Yaskawa INFORM job: A_ROOF_SIDE_0617_2_PAINT_6.JBI

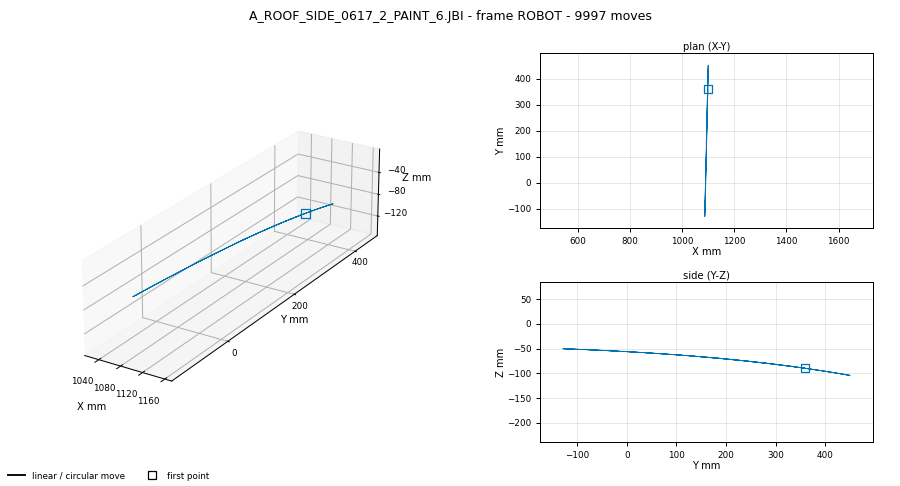
[picture p0: tool path of A_ROOF_SIDE_0617_2_PAINT_6.JBI in frame ROBOT, 9997 of 9997 moves have a stored position in this frame; points joined in program order, loops and branches not executed]
/JOB
//NAME A_ROOF_SIDE_0617_2_PAINT6
//POS
///NPOS 9997,0,0,0,0,0
///TOOL 1
///USER 0
///POSTYPE ROBOT
///RECTAN
///RCONF 1,0,0,0,0,0,0,0,0,0,0,0,0,0,0,0,0,0,0,0,0,0,0,0
C00000=1098.381,359.221,-89.235,178.998,19.661,152.457
C00001=1098.376,358.973,-89.200,178.995,19.657,152.456
C00002=1098.369,358.726,-89.165,178.993,19.653,152.456
C00003=1098.364,358.478,-89.130,178.990,19.649,152.455
C00004=1098.358,358.230,-89.095,178.986,19.645,152.455
C00005=1098.352,357.983,-89.061,178.984,19.641,152.455
C00006=1098.347,357.735,-89.026,178.980,19.637,152.454
C00007=1098.340,357.488,-88.991,178.977,19.632,152.454
C00008=1098.332,357.110,-88.938,178.973,19.626,152.453
C00009=1098.324,356.733,-88.885,178.968,19.620,152.452
C00010=1098.314,356.355,-88.832,178.964,19.614,152.452
C00011=1098.306,355.978,-88.780,178.959,19.608,152.451
C00012=1098.300,355.731,-88.744,178.956,19.604,152.451
C00013=1098.295,355.483,-88.709,178.953,19.600,152.450
C00014=1098.289,355.235,-88.675,178.950,19.596,152.450
C00015=1098.284,354.988,-88.641,178.947,19.592,152.449
C00016=1098.277,354.740,-88.605,178.944,19.588,152.449
C00017=1098.272,354.493,-88.571,178.941,19.585,152.449
C00018=1098.266,354.245,-88.537,178.938,19.580,152.448
C00019=1098.261,353.998,-88.502,178.935,19.576,152.448
C00020=1098.254,353.750,-88.468,178.932,19.572,152.447
C00021=1098.249,353.502,-88.433,178.929,19.568,152.447
C00022=1098.243,353.255,-88.399,178.926,19.565,152.446
C00023=1098.237,353.007,-88.364,178.923,19.561,152.446
C00024=1098.231,352.760,-88.329,178.919,19.557,152.446
C00025=1098.226,352.513,-88.295,178.917,19.553,152.445
C00026=1098.220,352.265,-88.260,178.913,19.549,152.445
C00027=1098.214,352.017,-88.226,178.911,19.545,152.445
C00028=1098.208,351.770,-88.192,178.907,19.541,152.444
C00029=1098.203,351.522,-88.157,178.905,19.538,152.444
C00030=1098.197,351.275,-88.123,178.901,19.534,152.443
C00031=1098.191,351.027,-88.089,178.898,19.530,152.443
C00032=1098.186,350.779,-88.055,178.895,19.526,152.443
C00033=1098.180,350.531,-88.021,178.892,19.522,152.442
C00034=1098.174,350.284,-87.987,178.889,19.519,152.442
C00035=1098.169,350.037,-87.952,178.886,19.515,152.442
C00036=1098.163,349.789,-87.918,178.883,19.512,152.441
C00037=1098.157,349.541,-87.884,178.880,19.507,152.441
C00038=1098.151,349.294,-87.850,178.877,19.504,152.441
C00039=1098.146,349.046,-87.815,178.874,19.500,152.440
C00040=1098.140,348.799,-87.782,178.871,19.497,152.440
C00041=1098.134,348.551,-87.748,178.868,19.493,152.440
C00042=1098.128,348.303,-87.713,178.865,19.489,152.439
C00043=1098.123,348.056,-87.679,178.861,19.485,152.439
C00044=1098.117,347.808,-87.645,178.859,19.482,152.439
C00045=1098.111,347.561,-87.611,178.855,19.478,152.438
C00046=1098.105,347.313,-87.577,178.853,19.475,152.438
C00047=1098.100,347.066,-87.543,178.849,19.470,152.438
C00048=1098.095,346.818,-87.509,178.847,19.467,152.437
C00049=1098.088,346.570,-87.475,178.843,19.463,152.437
C00050=1098.082,346.322,-87.441,178.840,19.460,152.437
C00051=1098.077,346.075,-87.407,178.837,19.456,152.436
C00052=1098.071,345.827,-87.373,178.834,19.453,152.436
C00053=1098.065,345.579,-87.340,178.831,19.449,152.436
C00054=1098.060,345.332,-87.305,178.828,19.445,152.435
C00055=1098.054,345.084,-87.271,178.824,19.442,152.435
C00056=1098.049,344.837,-87.238,178.822,19.438,152.435
C00057=1098.043,344.589,-87.204,178.818,19.434,152.434
C00058=1098.038,344.341,-87.170,178.815,19.431,152.434
C00059=1098.031,344.093,-87.136,178.812,19.427,152.434
C00060=1098.022,343.718,-87.085,178.808,19.422,152.433
C00061=1098.014,343.343,-87.034,178.803,19.417,152.433
C00062=1098.005,342.968,-86.983,178.798,19.412,152.433
C00063=1097.996,342.593,-86.933,178.793,19.406,152.432
C00064=1097.990,342.345,-86.899,178.790,19.403,152.432
C00065=1097.984,342.098,-86.865,178.788,19.400,152.432
C00066=1097.979,341.850,-86.831,178.784,19.396,152.431
C00067=1097.973,341.602,-86.798,178.781,19.393,152.431
C00068=1097.967,341.354,-86.764,178.778,19.389,152.431
C00069=1097.962,341.107,-86.731,178.775,19.386,152.431
C00070=1097.956,340.859,-86.697,178.771,19.382,152.430
C00071=1097.951,340.611,-86.664,178.769,19.379,152.430
C00072=1097.945,340.363,-86.630,178.766,19.376,152.430
C00073=1097.939,340.116,-86.597,178.762,19.372,152.430
C00074=1097.934,339.868,-86.563,178.759,19.369,152.429
C00075=1097.928,339.620,-86.530,178.756,19.365,152.429
C00076=1097.922,339.373,-86.497,178.753,19.362,152.429
C00077=1097.917,339.126,-86.464,178.750,19.359,152.429
C00078=1097.911,338.878,-86.430,178.747,19.355,152.428
C00079=1097.906,338.630,-86.397,178.744,19.352,152.428
C00080=1097.900,338.382,-86.364,178.740,19.349,152.428
C00081=1097.894,338.134,-86.330,178.737,19.345,152.428
C00082=1097.888,337.887,-86.297,178.735,19.342,152.427
C00083=1097.882,337.639,-86.263,178.731,19.339,152.427
C00084=1097.877,337.391,-86.230,178.728,19.335,152.427
C00085=1097.871,337.143,-86.197,178.725,19.332,152.427
C00086=1097.865,336.896,-86.164,178.722,19.329,152.427
C00087=1097.859,336.648,-86.131,178.719,19.326,152.426
C00088=1097.854,336.400,-86.097,178.715,19.322,152.426
C00089=1097.847,336.152,-86.065,178.712,19.319,152.426
C00090=1097.842,335.904,-86.031,178.709,19.316,152.426
C00091=1097.836,335.656,-85.998,178.706,19.312,152.426
C00092=1097.831,335.409,-85.965,178.703,19.309,152.425
C00093=1097.825,335.162,-85.932,178.700,19.307,152.425
C00094=1097.820,334.914,-85.899,178.696,19.303,152.425
C00095=1097.814,334.666,-85.866,178.694,19.300,152.425
C00096=1097.808,334.418,-85.833,178.691,19.297,152.424
C00097=1097.802,334.170,-85.799,178.687,19.293,152.424
C00098=1097.797,333.922,-85.767,178.684,19.290,152.424
C00099=1097.791,333.674,-85.734,178.681,19.287,152.424
C00100=1097.786,333.427,-85.701,178.678,19.283,152.424
C00101=1097.779,333.179,-85.668,178.675,19.281,152.424
C00102=1097.774,332.932,-85.635,178.672,19.278,152.423
C00103=1097.769,332.683,-85.602,178.668,19.274,152.423
C00104=1097.762,332.435,-85.570,178.665,19.271,152.423
C00105=1097.757,332.187,-85.536,178.662,19.268,152.423
C00106=1097.751,331.941,-85.504,178.659,19.265,152.423
C00107=1097.745,331.693,-85.471,178.656,19.262,152.423
C00108=1097.739,331.444,-85.439,178.653,19.259,152.422
C00109=1097.734,331.197,-85.405,178.650,19.256,152.422
C00110=1097.728,330.949,-85.373,178.646,19.253,152.422
C00111=1097.722,330.701,-85.340,178.643,19.250,152.422
C00112=1097.713,330.320,-85.290,178.638,19.245,152.422
C00113=1097.704,329.938,-85.240,178.634,19.240,152.421
C00114=1097.695,329.558,-85.189,178.628,19.236,152.421
C00115=1097.686,329.176,-85.139,178.624,19.231,152.421
C00116=1097.680,328.929,-85.107,178.620,19.228,152.421
C00117=1097.675,328.680,-85.074,178.617,19.225,152.421
C00118=1097.669,328.432,-85.041,178.614,19.222,152.421
C00119=1097.663,328.185,-85.010,178.611,19.220,152.421
C00120=1097.658,327.937,-84.976,178.607,19.216,152.420
C00121=1097.652,327.689,-84.944,178.605,19.213,152.420
C00122=1097.645,327.441,-84.912,178.602,19.211,152.420
C00123=1097.640,327.194,-84.880,178.598,19.208,152.420
C00124=1097.634,326.946,-84.847,178.595,19.204,152.420
C00125=1097.628,326.698,-84.814,178.592,19.201,152.420
C00126=1097.622,326.450,-84.782,178.589,19.199,152.420
C00127=1097.618,326.202,-84.749,178.586,19.196,152.420
C00128=1097.612,325.954,-84.717,178.582,19.193,152.420
C00129=1097.605,325.706,-84.685,178.579,19.190,152.419
C00130=1097.600,325.459,-84.653,178.576,19.187,152.419
C00131=1097.595,325.210,-84.620,178.573,19.184,152.419
C00132=1097.588,324.963,-84.588,178.569,19.181,152.419
C00133=1097.583,324.715,-84.556,178.566,19.178,152.419
C00134=1097.577,324.467,-84.524,178.563,19.175,152.419
C00135=1097.571,324.219,-84.491,178.560,19.173,152.419
C00136=1097.566,323.972,-84.459,178.557,19.170,152.419
C00137=1097.560,323.723,-84.427,178.553,19.167,152.418
C00138=1097.554,323.475,-84.395,178.550,19.164,152.418
C00139=1097.548,323.228,-84.363,178.547,19.161,152.418
C00140=1097.543,322.980,-84.330,178.544,19.158,152.418
C00141=1097.538,322.732,-84.298,178.542,19.155,152.418
C00142=1097.532,322.484,-84.266,178.538,19.152,152.418
C00143=1097.526,322.236,-84.234,178.535,19.149,152.418
C00144=1097.520,321.989,-84.202,178.532,19.147,152.418
C00145=1097.514,321.741,-84.170,178.529,19.144,152.418
C00146=1097.509,321.493,-84.138,178.526,19.141,152.418
C00147=1097.503,321.245,-84.106,178.522,19.138,152.417
C00148=1097.497,320.996,-84.074,178.519,19.135,152.417
C00149=1097.492,320.749,-84.042,178.516,19.133,152.417
C00150=1097.486,320.501,-84.010,178.513,19.130,152.417
C00151=1097.481,320.253,-83.978,178.510,19.127,152.417
C00152=1097.475,320.005,-83.946,178.507,19.125,152.417
C00153=1097.469,319.757,-83.914,178.503,19.121,152.417
C00154=1097.464,319.509,-83.882,178.500,19.119,152.417
C00155=1097.459,319.261,-83.850,178.497,19.116,152.417
C00156=1097.453,319.013,-83.818,178.494,19.113,152.417
C00157=1097.447,318.766,-83.787,178.491,19.111,152.417
C00158=1097.441,318.517,-83.754,178.488,19.108,152.417
C00159=1097.436,318.270,-83.723,178.484,19.105,152.416
C00160=1097.430,318.022,-83.691,178.481,19.102,152.416
C00161=1097.425,317.774,-83.659,178.478,19.099,152.416
C00162=1097.419,317.527,-83.627,178.475,19.097,152.416
C00163=1097.413,317.279,-83.595,178.472,19.094,152.416
C00164=1097.405,316.890,-83.546,178.466,19.089,152.416
C00165=1097.397,316.502,-83.496,178.462,19.085,152.416
C00166=1097.387,316.114,-83.447,178.456,19.081,152.416
C00167=1097.379,315.725,-83.397,178.452,19.077,152.416
C00168=1097.373,315.478,-83.365,178.449,19.074,152.416
C00169=1097.368,315.229,-83.334,178.445,19.071,152.416
C00170=1097.362,314.981,-83.302,178.442,19.068,152.416
C00171=1097.356,314.734,-83.271,178.439,19.066,152.416
C00172=1097.350,314.486,-83.239,178.435,19.063,152.416
C00173=1097.344,314.237,-83.208,178.432,19.061,152.416
C00174=1097.338,313.990,-83.177,178.429,19.058,152.416
C00175=1097.332,313.742,-83.145,178.426,19.056,152.415
C00176=1097.327,313.494,-83.114,178.423,19.053,152.416
C00177=1097.321,313.246,-83.082,178.420,19.051,152.415
C00178=1097.315,312.998,-83.051,178.416,19.047,152.415
C00179=1097.310,312.750,-83.020,178.412,19.045,152.415
C00180=1097.303,312.502,-82.988,178.409,19.043,152.415
C00181=1097.298,312.255,-82.957,178.406,19.040,152.415
C00182=1097.292,312.006,-82.925,178.403,19.038,152.415
C00183=1097.286,311.759,-82.894,178.400,19.035,152.415
C00184=1097.280,311.510,-82.863,178.397,19.033,152.415
C00185=1097.275,311.262,-82.831,178.394,19.030,152.415
C00186=1097.269,311.014,-82.801,178.391,19.028,152.415
C00187=1097.263,310.766,-82.769,178.387,19.025,152.415
C00188=1097.257,310.518,-82.739,178.384,19.023,152.415
C00189=1097.252,310.271,-82.707,178.380,19.020,152.415
C00190=1097.246,310.022,-82.676,178.377,19.017,152.415
C00191=1097.240,309.775,-82.645,178.374,19.015,152.415
C00192=1097.235,309.527,-82.614,178.371,19.013,152.415
C00193=1097.228,309.279,-82.582,178.367,19.010,152.415
C00194=1097.223,309.031,-82.551,178.364,19.008,152.415
C00195=1097.217,308.783,-82.520,178.361,19.005,152.415
C00196=1097.212,308.535,-82.489,178.358,19.003,152.415
C00197=1097.207,308.287,-82.458,178.355,19.000,152.415
C00198=1097.200,308.039,-82.427,178.352,18.998,152.415
C00199=1097.195,307.791,-82.396,178.348,18.996,152.416
C00200=1097.189,307.543,-82.365,178.345,18.993,152.415
C00201=1097.183,307.295,-82.334,178.342,18.991,152.415
C00202=1097.178,307.047,-82.303,178.339,18.988,152.415
C00203=1097.173,306.799,-82.272,178.335,18.985,152.416
C00204=1097.166,306.551,-82.242,178.332,18.983,152.416
C00205=1097.161,306.303,-82.210,178.329,18.980,152.415
C00206=1097.155,306.055,-82.180,178.325,18.978,152.416
C00207=1097.150,305.807,-82.149,178.322,18.975,152.415
C00208=1097.143,305.559,-82.118,178.319,18.973,152.416
C00209=1097.138,305.311,-82.086,178.316,18.971,152.416
C00210=1097.132,305.063,-82.056,178.313,18.968,152.416
C00211=1097.127,304.815,-82.025,178.309,18.966,152.416
C00212=1097.121,304.567,-81.995,178.306,18.963,152.416
C00213=1097.116,304.320,-81.964,178.303,18.961,152.416
C00214=1097.110,304.071,-81.933,178.300,18.958,152.416
C00215=1097.104,303.824,-81.902,178.297,18.956,152.416
C00216=1097.096,303.437,-81.855,178.291,18.952,152.416
C00217=1097.087,303.052,-81.807,178.286,18.948,152.416
C00218=1097.077,302.666,-81.759,178.281,18.945,152.416
C00219=1097.069,302.281,-81.711,178.277,18.941,152.416
C00220=1097.064,302.032,-81.680,178.273,18.939,152.416
C00221=1097.058,301.785,-81.650,178.270,18.936,152.416
C00222=1097.052,301.537,-81.619,178.267,18.934,152.416
C00223=1097.047,301.289,-81.588,178.264,18.932,152.416
C00224=1097.041,301.041,-81.558,178.260,18.928,152.416
C00225=1097.036,300.793,-81.528,178.257,18.926,152.416
C00226=1097.031,300.545,-81.497,178.253,18.924,152.416
C00227=1097.025,300.296,-81.467,178.250,18.922,152.416
C00228=1097.019,300.049,-81.437,178.247,18.919,152.416
C00229=1097.014,299.801,-81.406,178.244,18.917,152.416
C00230=1097.008,299.553,-81.376,178.240,18.914,152.416
C00231=1097.002,299.305,-81.345,178.237,18.912,152.416
C00232=1096.997,299.057,-81.314,178.234,18.910,152.416
C00233=1096.992,298.809,-81.284,178.231,18.907,152.416
C00234=1096.986,298.560,-81.254,178.228,18.905,152.416
C00235=1096.981,298.312,-81.223,178.224,18.903,152.416
C00236=1096.975,298.065,-81.193,178.221,18.900,152.417
C00237=1096.969,297.816,-81.162,178.218,18.898,152.417
C00238=1096.963,297.568,-81.133,178.214,18.896,152.417
C00239=1096.957,297.320,-81.102,178.211,18.894,152.417
C00240=1096.952,297.072,-81.072,178.208,18.891,152.417
C00241=1096.947,296.824,-81.041,178.205,18.889,152.417
C00242=1096.941,296.575,-81.011,178.202,18.887,152.417
C00243=1096.935,296.328,-80.981,178.199,18.885,152.417
C00244=1096.929,296.080,-80.951,178.196,18.883,152.417
C00245=1096.924,295.831,-80.921,178.193,18.880,152.417
C00246=1096.918,295.583,-80.891,178.189,18.878,152.417
C00247=1096.912,295.336,-80.860,178.186,18.876,152.417
C00248=1096.907,295.087,-80.831,178.183,18.874,152.417
C00249=1096.901,294.839,-80.800,178.179,18.871,152.417
C00250=1096.895,294.591,-80.771,178.176,18.869,152.418
C00251=1096.890,294.343,-80.740,178.173,18.867,152.418
C00252=1096.884,294.095,-80.711,178.169,18.865,152.418
C00253=1096.878,293.847,-80.680,178.166,18.863,152.418
C00254=1096.872,293.599,-80.650,178.163,18.860,152.418
C00255=1096.867,293.351,-80.620,178.160,18.858,152.418
C00256=1096.861,293.103,-80.590,178.156,18.856,152.418
C00257=1096.856,292.854,-80.560,178.153,18.854,152.418
C00258=1096.850,292.606,-80.531,178.150,18.851,152.418
C00259=1096.844,292.358,-80.500,178.146,18.849,152.418
C00260=1096.839,292.110,-80.471,178.143,18.847,152.418
C00261=1096.833,291.862,-80.440,178.140,18.845,152.418
C00262=1096.828,291.614,-80.411,178.137,18.842,152.419
C00263=1096.822,291.366,-80.381,178.134,18.841,152.419
C00264=1096.816,291.118,-80.352,178.131,18.839,152.419
C00265=1096.810,290.870,-80.322,178.127,18.837,152.419
C00266=1096.805,290.622,-80.292,178.124,18.834,152.419
C00267=1096.799,290.373,-80.262,178.121,18.832,152.419
C00268=1096.791,290.001,-80.217,178.116,18.829,152.419
C00269=1096.782,289.630,-80.173,178.111,18.826,152.419
C00270=1096.774,289.258,-80.128,178.106,18.822,152.420
C00271=1096.765,288.887,-80.084,178.101,18.819,152.420
C00272=1096.759,288.638,-80.054,178.098,18.817,152.420
C00273=1096.754,288.390,-80.025,178.095,18.815,152.420
C00274=1096.748,288.141,-79.995,178.092,18.813,152.420
C00275=1096.742,287.894,-79.965,178.088,18.811,152.420
C00276=1096.736,287.645,-79.936,178.085,18.809,152.420
C00277=1096.731,287.398,-79.906,178.082,18.807,152.420
C00278=1096.726,287.149,-79.877,178.078,18.805,152.420
C00279=1096.720,286.901,-79.848,178.075,18.802,152.421
C00280=1096.714,286.653,-79.818,178.071,18.801,152.421
C00281=1096.709,286.404,-79.789,178.068,18.798,152.421
C00282=1096.702,286.157,-79.759,178.066,18.797,152.421
C00283=1096.697,285.909,-79.730,178.062,18.794,152.421
C00284=1096.692,285.660,-79.700,178.059,18.793,152.421
C00285=1096.685,285.412,-79.671,178.056,18.790,152.421
C00286=1096.680,285.164,-79.641,178.052,18.788,152.421
C00287=1096.674,284.915,-79.612,178.049,18.786,152.422
C00288=1096.669,284.668,-79.583,178.046,18.784,152.422
C00289=1096.663,284.420,-79.553,178.042,18.782,152.422
C00290=1096.658,284.171,-79.524,178.040,18.780,152.422
C00291=1096.651,283.923,-79.495,178.036,18.778,152.422
C00292=1096.646,283.675,-79.465,178.033,18.776,152.422
C00293=1096.641,283.427,-79.436,178.030,18.774,152.422
C00294=1096.635,283.179,-79.407,178.026,18.772,152.422
C00295=1096.629,282.930,-79.377,178.023,18.770,152.423
C00296=1096.624,282.681,-79.348,178.020,18.767,152.423
C00297=1096.618,282.434,-79.319,178.016,18.766,152.423
C00298=1096.613,282.185,-79.290,178.014,18.764,152.423
C00299=1096.607,281.937,-79.261,178.010,18.762,152.423
C00300=1096.602,281.689,-79.231,178.007,18.760,152.423
C00301=1096.595,281.441,-79.202,178.004,18.758,152.423
C00302=1096.590,281.193,-79.173,178.000,18.755,152.423
C00303=1096.584,280.944,-79.144,177.997,18.754,152.424
C00304=1096.579,280.696,-79.115,177.994,18.751,152.424
C00305=1096.573,280.448,-79.086,177.991,18.750,152.424
C00306=1096.567,280.200,-79.057,177.988,18.748,152.424
C00307=1096.561,279.951,-79.028,177.984,18.746,152.424
C00308=1096.556,279.703,-78.999,177.981,18.744,152.424
C00309=1096.550,279.455,-78.970,177.977,18.741,152.424
C00310=1096.545,279.207,-78.940,177.974,18.740,152.425
C00311=1096.539,278.959,-78.912,177.971,18.738,152.425
C00312=1096.533,278.711,-78.883,177.968,18.736,152.425
C00313=1096.528,278.462,-78.854,177.965,18.734,152.425
C00314=1096.522,278.214,-78.826,177.961,18.732,152.425
C00315=1096.517,277.966,-78.796,177.958,18.730,152.425
C00316=1096.511,277.717,-78.768,177.954,18.728,152.426
C00317=1096.505,277.469,-78.739,177.952,18.726,152.426
C00318=1096.500,277.221,-78.709,177.948,18.724,152.426
C00319=1096.494,276.972,-78.681,177.945,18.722,152.426
C00320=1096.486,276.610,-78.639,177.940,18.719,152.426
C00321=1096.478,276.248,-78.597,177.936,18.717,152.427
C00322=1096.469,275.885,-78.555,177.931,18.714,152.427
C00323=1096.460,275.523,-78.513,177.926,18.711,152.427
C00324=1096.456,275.275,-78.485,177.923,18.709,152.427
C00325=1096.450,275.026,-78.455,177.920,18.707,152.427
C00326=1096.444,274.778,-78.427,177.916,18.705,152.427
C00327=1096.439,274.530,-78.398,177.913,18.703,152.428
C00328=1096.433,274.281,-78.370,177.910,18.702,152.428
C00329=1096.427,274.034,-78.341,177.907,18.700,152.428
C00330=1096.421,273.785,-78.313,177.903,18.698,152.428
C00331=1096.416,273.536,-78.284,177.900,18.696,152.428
C00332=1096.410,273.289,-78.255,177.896,18.694,152.428
C00333=1096.404,273.040,-78.227,177.894,18.692,152.429
C00334=1096.399,272.792,-78.198,177.890,18.690,152.429
C00335=1096.393,272.544,-78.170,177.887,18.688,152.429
C00336=1096.388,272.295,-78.141,177.884,18.686,152.429
C00337=1096.382,272.046,-78.113,177.881,18.685,152.429
C00338=1096.376,271.798,-78.084,177.877,18.683,152.430
C00339=1096.371,271.550,-78.056,177.874,18.681,152.430
C00340=1096.365,271.302,-78.027,177.871,18.679,152.430
C00341=1096.359,271.054,-77.999,177.867,18.677,152.430
C00342=1096.353,270.805,-77.970,177.865,18.676,152.430
C00343=1096.349,270.557,-77.942,177.861,18.674,152.430
C00344=1096.343,270.308,-77.914,177.858,18.671,152.430
C00345=1096.337,270.060,-77.886,177.854,18.670,152.431
C00346=1096.331,269.812,-77.857,177.852,18.668,152.431
C00347=1096.326,269.564,-77.829,177.848,18.666,152.431
C00348=1096.320,269.315,-77.800,177.845,18.664,152.431
C00349=1096.314,269.067,-77.772,177.841,18.663,152.431
C00350=1096.308,268.818,-77.744,177.838,18.660,152.432
C00351=1096.303,268.570,-77.716,177.835,18.659,152.432
C00352=1096.297,268.322,-77.688,177.832,18.657,152.432
C00353=1096.292,268.074,-77.659,177.828,18.655,152.432
C00354=1096.286,267.825,-77.631,177.825,18.653,152.432
C00355=1096.280,267.577,-77.603,177.822,18.652,152.433
C00356=1096.274,267.329,-77.574,177.819,18.650,152.433
C00357=1096.269,267.081,-77.546,177.815,18.648,152.433
C00358=1096.263,266.832,-77.518,177.812,18.646,152.433
C00359=1096.258,266.584,-77.490,177.809,18.644,152.433
C00360=1096.252,266.335,-77.462,177.806,18.643,152.433
C00361=1096.246,266.087,-77.434,177.802,18.641,152.434
C00362=1096.241,265.839,-77.406,177.799,18.639,152.434
C00363=1096.235,265.590,-77.378,177.796,18.637,152.434
C00364=1096.230,265.342,-77.350,177.793,18.636,152.434
C00365=1096.224,265.093,-77.322,177.789,18.634,152.434
C00366=1096.219,264.845,-77.294,177.786,18.631,152.435
C00367=1096.213,264.597,-77.266,177.783,18.630,152.435
C00368=1096.207,264.348,-77.238,177.780,18.628,152.435
C00369=1096.201,264.100,-77.210,177.776,18.627,152.435
C00370=1096.195,263.851,-77.182,177.773,18.625,152.435
C00371=1096.190,263.603,-77.154,177.770,18.623,152.436
C00372=1096.182,263.243,-77.115,177.765,18.621,152.436
C00373=1096.173,262.884,-77.074,177.760,18.618,152.436
C00374=1096.165,262.525,-77.034,177.756,18.616,152.437
C00375=1096.157,262.164,-76.994,177.751,18.613,152.437
C00376=1096.151,261.916,-76.966,177.748,18.612,152.437
C00377=1096.145,261.668,-76.938,177.745,18.610,152.437
C00378=1096.139,261.420,-76.910,177.741,18.608,152.438
C00379=1096.134,261.171,-76.883,177.738,18.606,152.438
C00380=1096.128,260.923,-76.855,177.735,18.605,152.438
C00381=1096.122,260.674,-76.827,177.731,18.603,152.438
C00382=1096.116,260.426,-76.799,177.728,18.602,152.439
C00383=1096.111,260.178,-76.772,177.725,18.600,152.439
C00384=1096.105,259.929,-76.744,177.722,18.598,152.439
C00385=1096.100,259.680,-76.717,177.718,18.596,152.439
C00386=1096.094,259.432,-76.689,177.716,18.595,152.439
C00387=1096.088,259.184,-76.661,177.712,18.593,152.440
C00388=1096.083,258.935,-76.634,177.709,18.591,152.440
C00389=1096.076,258.687,-76.606,177.705,18.590,152.440
C00390=1096.071,258.438,-76.579,177.702,18.588,152.440
C00391=1096.065,258.190,-76.551,177.699,18.586,152.440
C00392=1096.060,257.942,-76.524,177.695,18.584,152.441
C00393=1096.054,257.693,-76.496,177.693,18.583,152.441
C00394=1096.048,257.445,-76.469,177.689,18.581,152.441
C00395=1096.043,257.196,-76.441,177.686,18.580,152.441
C00396=1096.037,256.948,-76.415,177.683,18.578,152.442
C00397=1096.031,256.699,-76.386,177.679,18.576,152.442
C00398=1096.026,256.451,-76.359,177.676,18.575,152.442
C00399=1096.020,256.203,-76.332,177.673,18.573,152.442
C00400=1096.015,255.954,-76.305,177.670,18.571,152.442
C00401=1096.008,255.706,-76.277,177.666,18.569,152.443
C00402=1096.003,255.457,-76.250,177.664,18.568,152.443
C00403=1095.997,255.209,-76.223,177.660,18.566,152.443
C00404=1095.992,254.961,-76.195,177.657,18.565,152.443
C00405=1095.986,254.712,-76.168,177.654,18.563,152.444
C00406=1095.980,254.464,-76.140,177.650,18.562,152.444
C00407=1095.974,254.215,-76.113,177.647,18.560,152.444
C00408=1095.969,253.966,-76.086,177.644,18.558,152.444
C00409=1095.963,253.719,-76.059,177.641,18.556,152.444
C00410=1095.958,253.469,-76.031,177.637,18.554,152.445
C00411=1095.952,253.221,-76.004,177.635,18.553,152.445
C00412=1095.947,252.972,-75.977,177.631,18.551,152.445
C00413=1095.941,252.725,-75.950,177.628,18.550,152.445
C00414=1095.936,252.476,-75.923,177.625,18.548,152.446
C00415=1095.930,252.228,-75.896,177.621,18.547,152.446
C00416=1095.924,251.978,-75.868,177.618,18.544,152.446
C00417=1095.919,251.730,-75.842,177.615,18.543,152.446
C00418=1095.913,251.482,-75.814,177.612,18.541,152.446
C00419=1095.908,251.233,-75.787,177.608,18.540,152.447
C00420=1095.902,250.985,-75.760,177.606,18.538,152.447
C00421=1095.897,250.736,-75.733,177.602,18.536,152.447
C00422=1095.892,250.488,-75.706,177.598,18.535,152.447
C00423=1095.886,250.239,-75.679,177.596,18.533,152.448
C00424=1095.877,249.877,-75.639,177.591,18.531,152.448
C00425=1095.869,249.514,-75.600,177.586,18.528,152.448
C00426=1095.862,249.152,-75.561,177.582,18.526,152.448
C00427=1095.853,248.789,-75.521,177.576,18.523,152.449
C00428=1095.847,248.540,-75.494,177.574,18.522,152.449
C00429=1095.842,248.292,-75.468,177.570,18.520,152.449
C00430=1095.837,248.043,-75.441,177.567,18.518,152.449
C00431=1095.831,247.795,-75.414,177.564,18.517,152.450
C00432=1095.826,247.546,-75.387,177.561,18.515,152.450
C00433=1095.820,247.298,-75.360,177.558,18.514,152.450
C00434=1095.814,247.050,-75.333,177.554,18.512,152.450
C00435=1095.809,246.801,-75.307,177.551,18.510,152.451
C00436=1095.804,246.553,-75.279,177.548,18.509,152.451
C00437=1095.798,246.304,-75.253,177.545,18.507,152.451
C00438=1095.792,246.055,-75.227,177.541,18.505,152.451
C00439=1095.786,245.807,-75.200,177.538,18.504,152.452
C00440=1095.781,245.559,-75.174,177.535,18.502,152.452
C00441=1095.776,245.310,-75.146,177.532,18.501,152.452
C00442=1095.770,245.062,-75.120,177.529,18.499,152.452
C00443=1095.764,244.813,-75.093,177.525,18.498,152.453
C00444=1095.758,244.565,-75.066,177.522,18.496,152.453
C00445=1095.753,244.316,-75.040,177.519,18.495,152.453
C00446=1095.748,244.067,-75.013,177.516,18.493,152.453
C00447=1095.742,243.819,-74.987,177.513,18.492,152.454
C00448=1095.736,243.570,-74.960,177.509,18.490,152.454
C00449=1095.731,243.321,-74.934,177.506,18.489,152.454
C00450=1095.725,243.073,-74.907,177.503,18.487,152.454
C00451=1095.719,242.825,-74.881,177.500,18.486,152.454
C00452=1095.714,242.576,-74.854,177.497,18.484,152.455
C00453=1095.708,242.327,-74.828,177.493,18.482,152.455
C00454=1095.702,242.079,-74.801,177.490,18.481,152.455
C00455=1095.697,241.831,-74.775,177.487,18.479,152.455
C00456=1095.691,241.582,-74.749,177.484,18.478,152.456
C00457=1095.685,241.333,-74.722,177.481,18.476,152.456
C00458=1095.679,241.085,-74.696,177.478,18.475,152.456
C00459=1095.674,240.836,-74.670,177.474,18.473,152.456
C00460=1095.668,240.588,-74.643,177.471,18.471,152.457
C00461=1095.663,240.339,-74.617,177.468,18.470,152.457
C00462=1095.657,240.090,-74.590,177.465,18.468,152.457
C00463=1095.651,239.842,-74.564,177.462,18.467,152.457
C00464=1095.646,239.593,-74.538,177.458,18.466,152.458
C00465=1095.640,239.345,-74.511,177.454,18.464,152.458
C00466=1095.635,239.096,-74.485,177.452,18.462,152.458
C00467=1095.629,238.847,-74.459,177.448,18.461,152.459
C00468=1095.623,238.598,-74.433,177.446,18.459,152.459
C00469=1095.618,238.350,-74.406,177.442,18.458,152.459
C00470=1095.613,238.102,-74.380,177.439,18.456,152.459
C00471=1095.607,237.853,-74.354,177.436,18.455,152.460
C00472=1095.601,237.604,-74.328,177.433,18.453,152.460
C00473=1095.595,237.356,-74.302,177.429,18.452,152.460
C00474=1095.589,237.107,-74.276,177.426,18.450,152.460
C00475=1095.584,236.858,-74.250,177.423,18.449,152.460
C00476=1095.576,236.489,-74.211,177.419,18.447,152.461
C00477=1095.567,236.120,-74.173,177.413,18.444,152.461
C00478=1095.559,235.751,-74.133,177.409,18.442,152.462
C00479=1095.551,235.381,-74.095,177.404,18.440,152.462
C00480=1095.545,235.133,-74.069,177.401,18.438,152.462
C00481=1095.540,234.884,-74.043,177.398,18.437,152.463
C00482=1095.534,234.635,-74.017,177.394,18.435,152.463
C00483=1095.529,234.386,-73.991,177.392,18.434,152.463
C00484=1095.523,234.138,-73.965,177.388,18.432,152.463
C00485=1095.517,233.889,-73.939,177.385,18.431,152.464
C00486=1095.512,233.640,-73.913,177.382,18.429,152.464
C00487=1095.506,233.392,-73.887,177.378,18.427,152.464
C00488=1095.500,233.143,-73.861,177.375,18.427,152.464
C00489=1095.495,232.895,-73.836,177.372,18.425,152.465
C00490=1095.489,232.646,-73.810,177.369,18.424,152.465
C00491=1095.484,232.397,-73.784,177.366,18.422,152.465
C00492=1095.478,232.149,-73.758,177.363,18.421,152.465
C00493=1095.472,231.900,-73.732,177.359,18.419,152.466
C00494=1095.467,231.652,-73.706,177.357,18.418,152.466
C00495=1095.461,231.403,-73.681,177.353,18.416,152.466
C00496=1095.456,231.154,-73.655,177.350,18.415,152.466
C00497=1095.450,230.905,-73.629,177.347,18.413,152.467
C00498=1095.445,230.657,-73.603,177.344,18.412,152.467
C00499=1095.439,230.408,-73.578,177.340,18.410,152.467
C00500=1095.433,230.159,-73.552,177.338,18.409,152.468
C00501=1095.427,229.911,-73.526,177.334,18.407,152.468
C00502=1095.422,229.663,-73.501,177.331,18.406,152.468
C00503=1095.416,229.414,-73.475,177.328,18.404,152.468
C00504=1095.410,229.165,-73.449,177.325,18.404,152.469
C00505=1095.404,228.917,-73.424,177.321,18.402,152.469
C00506=1095.399,228.668,-73.398,177.319,18.401,152.469
C00507=1095.394,228.419,-73.372,177.315,18.399,152.469
C00508=1095.388,228.171,-73.347,177.312,18.398,152.470
C00509=1095.382,227.922,-73.321,177.309,18.396,152.470
C00510=1095.377,227.674,-73.296,177.306,18.395,152.470
C00511=1095.371,227.425,-73.270,177.302,18.393,152.471
C00512=1095.365,227.176,-73.246,177.300,18.392,152.471
C00513=1095.360,226.927,-73.220,177.296,18.390,152.471
C00514=1095.354,226.679,-73.195,177.293,18.389,152.471
C00515=1095.349,226.430,-73.169,177.290,18.387,152.472
C00516=1095.343,226.182,-73.144,177.287,18.386,152.472
C00517=1095.337,225.933,-73.119,177.283,18.385,152.472
C00518=1095.331,225.684,-73.093,177.281,18.383,152.472
C00519=1095.326,225.436,-73.068,177.277,18.382,152.473
C00520=1095.321,225.186,-73.042,177.274,18.380,152.473
C00521=1095.314,224.938,-73.017,177.271,18.379,152.473
C00522=1095.310,224.689,-72.991,177.268,18.378,152.474
C00523=1095.303,224.441,-72.966,177.264,18.376,152.474
C00524=1095.298,224.192,-72.940,177.262,18.375,152.474
C00525=1095.293,223.943,-72.916,177.258,18.373,152.474
C00526=1095.286,223.695,-72.891,177.255,18.372,152.475
C00527=1095.282,223.446,-72.865,177.252,18.370,152.475
C00528=1095.273,223.068,-72.826,177.247,18.368,152.475
C00529=1095.265,222.689,-72.789,177.243,18.366,152.476
C00530=1095.256,222.312,-72.750,177.238,18.364,152.476
C00531=1095.247,221.934,-72.712,177.233,18.362,152.477
C00532=1095.242,221.685,-72.686,177.230,18.360,152.477
C00533=1095.236,221.436,-72.662,177.227,18.360,152.477
C00534=1095.230,221.188,-72.637,177.224,18.358,152.477
C00535=1095.225,220.940,-72.612,177.221,18.357,152.478
C00536=1095.219,220.690,-72.586,177.217,18.355,152.478
C00537=1095.213,220.442,-72.561,177.214,18.354,152.478
C00538=1095.208,220.193,-72.537,177.211,18.352,152.479
C00539=1095.202,219.944,-72.512,177.208,18.351,152.479
C00540=1095.197,219.695,-72.487,177.205,18.349,152.479
C00541=1095.191,219.447,-72.461,177.202,18.348,152.479
C00542=1095.186,219.198,-72.437,177.198,18.347,152.480
C00543=1095.179,218.949,-72.412,177.195,18.345,152.480
C00544=1095.174,218.701,-72.388,177.193,18.344,152.480
C00545=1095.169,218.452,-72.362,177.189,18.342,152.480
C00546=1095.163,218.203,-72.337,177.186,18.342,152.481
C00547=1095.157,217.955,-72.312,177.183,18.340,152.481
C00548=1095.151,217.705,-72.287,177.180,18.339,152.481
C00549=1095.146,217.457,-72.262,177.176,18.337,152.482
C00550=1095.140,217.208,-72.238,177.174,18.336,152.482
C00551=1095.135,216.960,-72.212,177.171,18.335,152.482
C00552=1095.130,216.711,-72.188,177.167,18.333,152.483
C00553=1095.124,216.462,-72.163,177.164,18.332,152.483
C00554=1095.118,216.214,-72.138,177.161,18.330,152.483
C00555=1095.112,215.965,-72.114,177.158,18.329,152.483
C00556=1095.107,215.717,-72.089,177.154,18.328,152.484
C00557=1095.101,215.467,-72.064,177.152,18.326,152.484
C00558=1095.095,215.219,-72.040,177.149,18.325,152.484
C00559=1095.090,214.970,-72.014,177.145,18.323,152.484
C00560=1095.085,214.721,-71.990,177.143,18.322,152.485
C00561=1095.079,214.473,-71.965,177.139,18.321,152.485
C00562=1095.073,214.223,-71.941,177.136,18.320,152.485
C00563=1095.068,213.975,-71.916,177.133,18.319,152.486
C00564=1095.062,213.726,-71.891,177.130,18.317,152.486
C00565=1095.057,213.478,-71.867,177.127,18.316,152.486
C00566=1095.051,213.229,-71.843,177.124,18.314,152.486
C00567=1095.045,212.980,-71.817,177.121,18.313,152.487
C00568=1095.040,212.732,-71.793,177.118,18.312,152.487
C00569=1095.034,212.482,-71.768,177.114,18.310,152.487
C00570=1095.029,212.234,-71.744,177.112,18.309,152.487
C00571=1095.023,211.985,-71.720,177.108,18.307,152.488
C00572=1095.017,211.737,-71.695,177.105,18.306,152.488
C00573=1095.012,211.488,-71.670,177.102,18.305,152.488
C00574=1095.006,211.239,-71.646,177.099,18.303,152.489
C00575=1095.001,210.990,-71.622,177.096,18.302,152.489
C00576=1094.995,210.742,-71.597,177.092,18.301,152.489
C00577=1094.989,210.492,-71.573,177.090,18.300,152.490
C00578=1094.984,210.244,-71.548,177.087,18.298,152.490
C00579=1094.978,209.995,-71.525,177.083,18.297,152.490
C00580=1094.970,209.621,-71.488,177.079,18.295,152.490
C00581=1094.961,209.247,-71.451,177.074,18.293,152.491
C00582=1094.952,208.872,-71.415,177.070,18.291,152.491
C00583=1094.944,208.498,-71.378,177.065,18.289,152.492
C00584=1094.921,207.483,-71.280,177.011,18.266,152.497
C00585=1094.916,207.234,-71.256,177.008,18.266,152.497
C00586=1094.910,206.986,-71.232,177.005,18.265,152.498
C00587=1094.904,206.737,-71.207,177.002,18.265,152.498
C00588=1094.899,206.488,-71.184,176.998,18.264,152.499
C00589=1094.893,206.239,-71.160,176.995,18.264,152.499
C00590=1094.888,205.991,-71.136,176.991,18.263,152.500
C00591=1094.882,205.741,-71.111,176.988,18.262,152.500
C00592=1094.876,205.492,-71.088,176.985,18.262,152.501
C00593=1094.871,205.244,-71.064,176.982,18.262,152.501
C00594=1094.865,204.996,-71.040,176.979,18.261,152.502
C00595=1094.860,204.746,-71.017,176.975,18.261,152.502
C00596=1094.855,204.498,-70.993,176.972,18.261,152.503
C00597=1094.848,204.249,-70.969,176.969,18.260,152.503
C00598=1094.843,204.000,-70.945,176.966,18.260,152.504
C00599=1094.837,203.751,-70.921,176.963,18.259,152.504
C00600=1094.832,203.503,-70.897,176.960,18.259,152.505
C00601=1094.827,203.254,-70.874,176.956,18.258,152.505
C00602=1094.821,203.005,-70.850,176.953,18.258,152.506
C00603=1094.816,202.756,-70.826,176.949,18.257,152.506
C00604=1094.809,202.507,-70.802,176.946,18.256,152.507
C00605=1094.804,202.258,-70.779,176.943,18.256,152.507
C00606=1094.798,202.010,-70.755,176.940,18.256,152.508
C00607=1094.792,201.761,-70.732,176.937,18.255,152.508
C00608=1094.787,201.512,-70.708,176.933,18.255,152.509
C00609=1094.780,201.263,-70.684,176.930,18.255,152.509
C00610=1094.775,201.014,-70.660,176.927,18.254,152.510
C00611=1094.769,200.766,-70.637,176.924,18.254,152.510
C00612=1094.764,200.517,-70.614,176.921,18.253,152.511
C00613=1094.758,200.268,-70.590,176.917,18.253,152.511
C00614=1094.752,200.019,-70.567,176.914,18.253,152.512
C00615=1094.747,199.770,-70.544,176.911,18.252,152.512
C00616=1094.741,199.521,-70.519,176.908,18.252,152.513
C00617=1094.735,199.272,-70.496,176.905,18.251,152.514
C00618=1094.729,199.024,-70.472,176.902,18.251,152.514
C00619=1094.724,198.775,-70.449,176.898,18.250,152.514
C00620=1094.718,198.526,-70.426,176.895,18.250,152.515
C00621=1094.712,198.278,-70.402,176.892,18.249,152.515
C00622=1094.707,198.028,-70.379,176.889,18.249,152.516
C00623=1094.701,197.780,-70.355,176.886,18.249,152.517
C00624=1094.696,197.531,-70.332,176.882,18.248,152.517
C00625=1094.691,197.282,-70.309,176.879,18.247,152.517
C00626=1094.685,197.034,-70.285,176.875,18.247,152.518
C00627=1094.678,196.784,-70.262,176.872,18.246,152.518
C00628=1094.673,196.535,-70.238,176.869,18.246,152.519
C00629=1094.667,196.286,-70.215,176.866,18.245,152.519
C00630=1094.661,196.038,-70.191,176.863,18.245,152.520
C00631=1094.656,195.788,-70.168,176.860,18.245,152.520
C00632=1094.651,195.540,-70.145,176.857,18.244,152.521
C00633=1094.645,195.291,-70.122,176.853,18.244,152.521
C00634=1094.639,195.042,-70.098,176.851,18.243,152.522
C00635=1094.634,194.793,-70.075,176.847,18.243,152.522
C00636=1094.628,194.544,-70.052,176.844,18.243,152.523
C00637=1094.622,194.295,-70.029,176.841,18.242,152.523
C00638=1094.617,194.047,-70.006,176.838,18.242,152.524
C00639=1094.611,193.798,-69.982,176.835,18.241,152.524
C00640=1094.606,193.549,-69.959,176.832,18.241,152.525
C00641=1094.600,193.300,-69.936,176.829,18.240,152.525
C00642=1094.594,193.051,-69.913,176.825,18.240,152.526
C00643=1094.589,192.802,-69.889,176.822,18.239,152.526
C00644=1094.584,192.553,-69.866,176.819,18.239,152.527
C00645=1094.577,192.278,-69.841,176.816,18.238,152.527
C00646=1094.572,192.003,-69.816,176.812,18.237,152.528
C00647=1094.565,191.729,-69.790,176.809,18.237,152.528
C00648=1094.559,191.453,-69.765,176.806,18.237,152.529
C00649=1094.553,191.204,-69.742,176.803,18.236,152.529
C00650=1094.548,190.955,-69.719,176.799,18.236,152.530
C00651=1094.543,190.706,-69.695,176.796,18.235,152.530
C00652=1094.537,190.457,-69.672,176.793,18.235,152.531
C00653=1094.531,190.208,-69.649,176.790,18.234,152.531
C00654=1094.526,189.959,-69.626,176.787,18.234,152.532
C00655=1094.520,189.710,-69.603,176.784,18.233,152.532
C00656=1094.515,189.462,-69.581,176.781,18.233,152.533
C00657=1094.510,189.213,-69.557,176.778,18.232,152.533
C00658=1094.504,188.964,-69.534,176.774,18.232,152.534
C00659=1094.498,188.715,-69.511,176.771,18.231,152.534
C00660=1094.493,188.466,-69.488,176.768,18.230,152.534
C00661=1094.487,188.217,-69.465,176.765,18.230,152.535
C00662=1094.481,187.968,-69.443,176.762,18.229,152.535
C00663=1094.476,187.720,-69.420,176.759,18.229,152.536
C00664=1094.471,187.471,-69.396,176.756,18.228,152.536
C00665=1094.465,187.222,-69.373,176.753,18.228,152.537
C00666=1094.460,186.973,-69.351,176.750,18.227,152.537
C00667=1094.454,186.724,-69.328,176.747,18.227,152.538
C00668=1094.449,186.476,-69.306,176.744,18.226,152.538
C00669=1094.443,186.227,-69.283,176.740,18.226,152.539
C00670=1094.437,185.978,-69.260,176.737,18.225,152.539
C00671=1094.432,185.729,-69.237,176.734,18.224,152.539
C00672=1094.426,185.479,-69.215,176.731,18.224,152.540
C00673=1094.421,185.231,-69.192,176.728,18.223,152.540
C00674=1094.415,184.982,-69.169,176.725,18.223,152.541
C00675=1094.410,184.733,-69.146,176.722,18.222,152.541
C00676=1094.404,184.484,-69.124,176.719,18.222,152.542
C00677=1094.399,184.235,-69.101,176.716,18.221,152.542
C00678=1094.392,183.986,-69.079,176.713,18.221,152.543
C00679=1094.386,183.737,-69.056,176.710,18.220,152.543
C00680=1094.381,183.488,-69.033,176.706,18.220,152.544
C00681=1094.375,183.239,-69.010,176.703,18.219,152.544
C00682=1094.370,182.991,-68.988,176.700,18.219,152.545
C00683=1094.364,182.742,-68.966,176.697,18.218,152.545
C00684=1094.358,182.493,-68.943,176.694,18.218,152.545
C00685=1094.352,182.244,-68.920,176.692,18.218,152.546
C00686=1094.347,181.995,-68.897,176.689,18.217,152.546
C00687=1094.341,181.746,-68.876,176.685,18.217,152.547
C00688=1094.335,181.498,-68.853,176.682,18.216,152.547
C00689=1094.330,181.248,-68.831,176.679,18.216,152.548
C00690=1094.324,180.999,-68.808,176.676,18.215,152.548
C00691=1094.318,180.751,-68.786,176.673,18.215,152.549
C00692=1094.312,180.501,-68.763,176.670,18.214,152.549
C00693=1094.307,180.252,-68.741,176.667,18.213,152.550
C00694=1094.301,180.004,-68.719,176.664,18.213,152.550
C00695=1094.295,179.755,-68.696,176.661,18.213,152.551
C00696=1094.290,179.505,-68.674,176.657,18.212,152.551
C00697=1094.283,179.257,-68.652,176.654,18.212,152.552
C00698=1094.278,179.008,-68.629,176.651,18.211,152.552
C00699=1094.273,178.759,-68.607,176.648,18.211,152.553
C00700=1094.267,178.510,-68.584,176.645,18.210,152.553
C00701=1094.261,178.261,-68.562,176.642,18.209,152.553
C00702=1094.256,178.012,-68.540,176.640,18.209,152.554
C00703=1094.250,177.763,-68.518,176.637,18.209,152.554
C00704=1094.244,177.514,-68.496,176.634,18.208,152.555
C00705=1094.239,177.265,-68.473,176.631,18.208,152.555
C00706=1094.233,177.017,-68.452,176.628,18.207,152.556
C00707=1094.227,176.768,-68.429,176.625,18.206,152.556
C00708=1094.222,176.518,-68.407,176.621,18.206,152.557
C00709=1094.215,176.243,-68.382,176.618,18.205,152.557
C00710=1094.210,175.967,-68.358,176.615,18.205,152.558
C00711=1094.203,175.692,-68.333,176.611,18.204,152.558
C00712=1094.197,175.416,-68.309,176.608,18.204,152.559
C00713=1094.191,175.167,-68.286,176.605,18.203,152.559
C00714=1094.185,174.918,-68.264,176.602,18.202,152.559
C00715=1094.181,174.669,-68.242,176.599,18.202,152.560
C00716=1094.174,174.421,-68.220,176.596,18.201,152.560
C00717=1094.169,174.172,-68.198,176.593,18.201,152.561
C00718=1094.163,173.922,-68.176,176.591,18.200,152.561
C00719=1094.157,173.674,-68.153,176.588,18.200,152.562
C00720=1094.153,173.425,-68.132,176.585,18.199,152.562
C00721=1094.146,173.176,-68.110,176.581,18.199,152.562
C00722=1094.141,172.926,-68.088,176.578,18.198,152.563
C00723=1094.135,172.678,-68.066,176.575,18.197,152.563
C00724=1094.130,172.429,-68.043,176.572,18.197,152.564
C00725=1094.124,172.179,-68.022,176.569,18.196,152.564
C00726=1094.119,171.931,-68.000,176.566,18.195,152.565
C00727=1094.112,171.682,-67.978,176.563,18.195,152.565
C00728=1094.107,171.433,-67.956,176.561,18.195,152.565
C00729=1094.102,171.184,-67.934,176.558,18.194,152.566
C00730=1094.096,170.935,-67.912,176.555,18.193,152.566
C00731=1094.091,170.686,-67.890,176.552,18.193,152.567
C00732=1094.085,170.436,-67.868,176.549,18.192,152.567
C00733=1094.080,170.188,-67.847,176.546,18.191,152.567
C00734=1094.074,169.939,-67.824,176.543,18.191,152.568
C00735=1094.069,169.690,-67.802,176.540,18.190,152.568
C00736=1094.063,169.441,-67.781,176.537,18.190,152.569
C00737=1094.058,169.192,-67.759,176.534,18.189,152.569
C00738=1094.052,168.943,-67.737,176.532,18.189,152.570
C00739=1094.047,168.694,-67.715,176.529,18.188,152.570
C00740=1094.041,168.445,-67.694,176.526,18.187,152.570
C00741=1094.036,168.196,-67.672,176.523,18.187,152.571
C00742=1094.030,167.947,-67.650,176.520,18.186,152.571
C00743=1094.025,167.698,-67.628,176.517,18.185,152.572
C00744=1094.019,167.449,-67.607,176.514,18.184,152.572
C00745=1094.014,167.200,-67.585,176.511,18.184,152.572
C00746=1094.008,166.951,-67.563,176.508,18.183,152.573
C00747=1094.003,166.702,-67.541,176.506,18.183,152.573
C00748=1093.997,166.453,-67.520,176.503,18.182,152.574
C00749=1093.992,166.204,-67.498,176.500,18.181,152.574
C00750=1093.986,165.955,-67.476,176.497,18.181,152.574
C00751=1093.980,165.706,-67.455,176.494,18.180,152.575
C00752=1093.975,165.457,-67.433,176.491,18.179,152.575
C00753=1093.969,165.208,-67.411,176.488,18.179,152.576
C00754=1093.964,164.959,-67.389,176.485,18.178,152.576
C00755=1093.958,164.710,-67.368,176.482,18.178,152.577
C00756=1093.953,164.462,-67.346,176.480,18.177,152.577
C00757=1093.947,164.212,-67.325,176.477,18.176,152.577
C00758=1093.942,163.963,-67.304,176.474,18.175,152.578
C00759=1093.936,163.714,-67.282,176.471,18.174,152.578
C00760=1093.931,163.465,-67.260,176.468,18.174,152.578
C00761=1093.926,163.216,-67.239,176.465,18.173,152.579
C00762=1093.920,162.967,-67.217,176.462,18.172,152.579
C00763=1093.915,162.718,-67.196,176.460,18.172,152.580
C00764=1093.909,162.469,-67.174,176.457,18.172,152.580
C00765=1093.904,162.220,-67.153,176.454,18.171,152.580
C00766=1093.899,161.971,-67.131,176.451,18.170,152.581
C00767=1093.893,161.721,-67.110,176.448,18.169,152.581
C00768=1093.887,161.473,-67.089,176.445,18.168,152.581
C00769=1093.881,161.224,-67.067,176.442,18.168,152.582
C00770=1093.876,160.975,-67.046,176.440,18.167,152.582
C00771=1093.871,160.726,-67.025,176.437,18.167,152.583
C00772=1093.865,160.477,-67.003,176.434,18.166,152.583
C00773=1093.858,160.201,-66.979,176.431,18.165,152.584
C00774=1093.853,159.926,-66.956,176.428,18.165,152.584
C00775=1093.846,159.649,-66.933,176.424,18.164,152.585
C00776=1093.840,159.373,-66.909,176.421,18.163,152.585
C00777=1093.834,159.125,-66.887,176.418,18.162,152.585
C00778=1093.828,158.875,-66.866,176.416,18.162,152.586
C00779=1093.823,158.626,-66.845,176.413,18.161,152.586
C00780=1093.817,158.378,-66.824,176.410,18.160,152.586
C00781=1093.811,158.128,-66.803,176.407,18.160,152.587
C00782=1093.807,157.879,-66.781,176.404,18.159,152.587
C00783=1093.801,157.629,-66.760,176.401,18.158,152.588
C00784=1093.795,157.381,-66.739,176.399,18.158,152.588
C00785=1093.790,157.132,-66.718,176.396,18.157,152.588
C00786=1093.784,156.883,-66.697,176.393,18.157,152.589
C00787=1093.778,156.634,-66.675,176.390,18.156,152.589
C00788=1093.773,156.385,-66.655,176.387,18.155,152.589
C00789=1093.767,156.136,-66.633,176.384,18.154,152.590
C00790=1093.762,155.887,-66.613,176.382,18.154,152.590
C00791=1093.756,155.638,-66.591,176.379,18.153,152.591
C00792=1093.750,155.388,-66.571,176.376,18.153,152.591
C00793=1093.745,155.140,-66.549,176.373,18.151,152.591
C00794=1093.739,154.891,-66.529,176.370,18.151,152.592
C00795=1093.733,154.641,-66.507,176.367,18.150,152.592
C00796=1093.728,154.392,-66.486,176.365,18.150,152.593
C00797=1093.722,154.144,-66.465,176.362,18.149,152.593
C00798=1093.717,153.894,-66.444,176.359,18.148,152.593
C00799=1093.711,153.645,-66.423,176.356,18.147,152.594
C00800=1093.706,153.396,-66.402,176.353,18.147,152.594
C00801=1093.700,153.147,-66.381,176.351,18.146,152.594
C00802=1093.694,152.898,-66.360,176.348,18.146,152.595
C00803=1093.689,152.649,-66.340,176.345,18.145,152.595
C00804=1093.683,152.400,-66.318,176.342,18.144,152.596
C00805=1093.678,152.151,-66.298,176.339,18.143,152.596
C00806=1093.672,151.901,-66.277,176.336,18.142,152.596
C00807=1093.667,151.653,-66.256,176.334,18.142,152.597
C00808=1093.661,151.403,-66.235,176.331,18.141,152.597
C00809=1093.655,151.155,-66.214,176.328,18.140,152.597
C00810=1093.649,150.906,-66.194,176.325,18.140,152.598
C00811=1093.644,150.657,-66.173,176.323,18.139,152.598
C00812=1093.638,150.407,-66.152,176.321,18.138,152.598
C00813=1093.633,150.158,-66.131,176.318,18.138,152.599
C00814=1093.627,149.909,-66.110,176.315,18.137,152.599
C00815=1093.622,149.660,-66.090,176.312,18.136,152.600
C00816=1093.617,149.412,-66.068,176.309,18.135,152.600
C00817=1093.610,149.162,-66.048,176.307,18.135,152.600
C00818=1093.605,148.913,-66.028,176.304,18.134,152.601
C00819=1093.600,148.664,-66.007,176.301,18.133,152.601
C00820=1093.594,148.415,-65.986,176.298,18.132,152.601
C00821=1093.588,148.166,-65.965,176.295,18.131,152.602
C00822=1093.582,147.917,-65.945,176.293,18.131,152.602
C00823=1093.577,147.668,-65.924,176.290,18.130,152.602
C00824=1093.572,147.418,-65.904,176.287,18.129,152.603
C00825=1093.565,147.169,-65.882,176.284,18.129,152.603
C00826=1093.559,146.920,-65.862,176.281,18.128,152.604
C00827=1093.554,146.671,-65.842,176.279,18.127,152.604
C00828=1093.549,146.422,-65.821,176.276,18.127,152.604
C00829=1093.543,146.173,-65.801,176.273,18.126,152.605
C00830=1093.537,145.924,-65.780,176.271,18.125,152.605
C00831=1093.532,145.674,-65.760,176.269,18.125,152.605
C00832=1093.526,145.426,-65.738,176.266,18.124,152.606
C00833=1093.520,145.177,-65.718,176.263,18.123,152.606
C00834=1093.515,144.928,-65.698,176.260,18.122,152.606
C00835=1093.510,144.679,-65.677,176.257,18.121,152.607
C00836=1093.503,144.429,-65.657,176.255,18.121,152.607
C00837=1093.497,144.154,-65.634,176.252,18.120,152.607
C00838=1093.491,143.877,-65.612,176.249,18.119,152.608
C00839=1093.486,143.601,-65.589,176.245,18.118,152.608
C00840=1093.479,143.325,-65.566,176.242,18.117,152.609
C00841=1093.473,143.076,-65.546,176.240,18.117,152.609
C00842=1093.468,142.827,-65.526,176.238,18.116,152.609
C00843=1093.463,142.577,-65.505,176.235,18.115,152.610
C00844=1093.457,142.329,-65.485,176.232,18.114,152.610
C00845=1093.451,142.079,-65.464,176.229,18.113,152.610
C00846=1093.445,141.830,-65.444,176.227,18.112,152.611
C00847=1093.440,141.581,-65.424,176.224,18.112,152.611
C00848=1093.434,141.332,-65.403,176.221,18.111,152.611
C00849=1093.428,141.083,-65.383,176.218,18.110,152.612
C00850=1093.423,140.834,-65.363,176.216,18.109,152.612
C00851=1093.418,140.585,-65.342,176.213,18.109,152.612
C00852=1093.412,140.336,-65.322,176.211,18.107,152.613
C00853=1093.407,140.087,-65.302,176.208,18.107,152.613
C00854=1093.401,139.837,-65.282,176.206,18.106,152.613
C00855=1093.396,139.588,-65.262,176.203,18.105,152.614
C00856=1093.389,139.339,-65.242,176.200,18.104,152.614
C00857=1093.384,139.090,-65.221,176.197,18.104,152.614
C00858=1093.378,138.841,-65.201,176.195,18.103,152.614
C00859=1093.372,138.592,-65.181,176.192,18.102,152.615
C00860=1093.366,138.343,-65.161,176.189,18.101,152.615
C00861=1093.362,138.093,-65.141,176.186,18.100,152.616
C00862=1093.356,137.844,-65.121,176.184,18.100,152.616
C00863=1093.350,137.595,-65.100,176.181,18.099,152.616
C00864=1093.344,137.346,-65.080,176.179,18.098,152.617
C00865=1093.339,137.097,-65.060,176.176,18.097,152.617
C00866=1093.333,136.848,-65.040,176.174,18.097,152.617
C00867=1093.327,136.599,-65.021,176.171,18.095,152.617
C00868=1093.322,136.350,-65.000,176.168,18.095,152.618
C00869=1093.316,136.101,-64.980,176.165,18.094,152.618
C00870=1093.311,135.851,-64.960,176.163,18.093,152.618
C00871=1093.305,135.602,-64.940,176.160,18.092,152.619
C00872=1093.299,135.354,-64.920,176.158,18.091,152.619
C00873=1093.294,135.104,-64.900,176.155,18.090,152.619
C00874=1093.288,134.855,-64.880,176.153,18.090,152.620
C00875=1093.283,134.606,-64.860,176.150,18.089,152.620
C00876=1093.277,134.357,-64.841,176.147,18.088,152.620
C00877=1093.271,134.108,-64.821,176.144,18.087,152.621
C00878=1093.266,133.859,-64.800,176.142,18.087,152.621
C00879=1093.260,133.609,-64.781,176.139,18.086,152.621
C00880=1093.255,133.360,-64.760,176.137,18.084,152.622
C00881=1093.249,133.111,-64.740,176.134,18.084,152.622
C00882=1093.243,132.862,-64.721,176.132,18.083,152.622
C00883=1093.238,132.613,-64.701,176.129,18.082,152.622
C00884=1093.232,132.363,-64.681,176.126,18.081,152.623
C00885=1093.226,132.114,-64.661,176.124,18.081,152.623
C00886=1093.221,131.865,-64.642,176.121,18.079,152.623
C00887=1093.216,131.616,-64.622,176.118,18.079,152.624
C00888=1093.210,131.367,-64.602,176.116,18.078,152.624
C00889=1093.204,131.118,-64.582,176.114,18.077,152.624
C00890=1093.198,130.869,-64.562,176.111,18.076,152.625
C00891=1093.192,130.619,-64.543,176.108,18.075,152.625
C00892=1093.187,130.370,-64.523,176.106,18.075,152.625
C00893=1093.181,130.121,-64.503,176.103,18.074,152.626
C00894=1093.175,129.872,-64.483,176.100,18.073,152.626
C00895=1093.170,129.623,-64.464,176.097,18.072,152.626
C00896=1093.164,129.374,-64.444,176.095,18.071,152.627
C00897=1093.158,129.124,-64.425,176.093,18.070,152.627
C00898=1093.153,128.875,-64.404,176.090,18.069,152.627
C00899=1093.147,128.626,-64.385,176.088,18.069,152.627
C00900=1093.141,128.376,-64.366,176.085,18.068,152.628
C00901=1093.134,128.101,-64.344,176.082,18.067,152.628
C00902=1093.128,127.824,-64.322,176.079,18.066,152.628
C00903=1093.122,127.548,-64.301,176.077,18.065,152.629
C00904=1093.116,127.272,-64.279,176.074,18.064,152.629
C00905=1093.110,127.022,-64.260,176.071,18.063,152.629
C00906=1093.104,126.774,-64.240,176.068,18.062,152.630
C00907=1093.099,126.524,-64.220,176.066,18.061,152.630
C00908=1093.093,126.275,-64.201,176.063,18.060,152.630
C00909=1093.087,126.026,-64.181,176.060,18.059,152.631
C00910=1093.081,125.777,-64.162,176.059,18.059,152.631
C00911=1093.076,125.527,-64.142,176.056,18.057,152.631
C00912=1093.071,125.279,-64.123,176.053,18.056,152.631
C00913=1093.065,125.029,-64.103,176.051,18.056,152.632
C00914=1093.060,124.780,-64.084,176.048,18.055,152.632
C00915=1093.054,124.531,-64.064,176.045,18.054,152.632
C00916=1093.048,124.282,-64.045,176.043,18.053,152.633
C00917=1093.042,124.032,-64.026,176.041,18.052,152.633
C00918=1093.037,123.783,-64.006,176.038,18.051,152.633
C00919=1093.031,123.535,-63.987,176.035,18.050,152.633
C00920=1093.026,123.285,-63.968,176.033,18.050,152.634
C00921=1093.020,123.036,-63.948,176.030,18.048,152.634
C00922=1093.014,122.786,-63.929,176.028,18.047,152.634
C00923=1093.008,122.538,-63.909,176.026,18.047,152.634
C00924=1093.003,122.289,-63.890,176.023,18.046,152.635
C00925=1092.997,122.039,-63.871,176.020,18.044,152.635
C00926=1092.992,121.790,-63.852,176.018,18.044,152.635
C00927=1092.986,121.540,-63.832,176.016,18.043,152.636
C00928=1092.980,121.291,-63.813,176.013,18.041,152.636
C00929=1092.975,121.043,-63.794,176.010,18.040,152.636
C00930=1092.969,120.794,-63.774,176.008,18.040,152.636
C00931=1092.964,120.544,-63.755,176.006,18.039,152.637
C00932=1092.958,120.295,-63.736,176.003,18.038,152.637
C00933=1092.953,120.046,-63.717,176.001,18.037,152.637
C00934=1092.947,119.796,-63.698,175.998,18.036,152.637
C00935=1092.941,119.547,-63.679,175.995,18.035,152.638
C00936=1092.936,119.298,-63.659,175.993,18.034,152.638
C00937=1092.931,119.049,-63.640,175.991,18.033,152.638
C00938=1092.925,118.799,-63.621,175.988,18.032,152.639
C00939=1092.919,118.550,-63.602,175.986,18.031,152.639
C00940=1092.914,118.301,-63.583,175.983,18.030,152.639
C00941=1092.908,118.052,-63.563,175.981,18.029,152.639
C00942=1092.903,117.803,-63.544,175.979,18.028,152.639
C00943=1092.897,117.554,-63.525,175.976,18.027,152.640
C00944=1092.892,117.305,-63.506,175.973,18.026,152.640
C00945=1092.886,117.055,-63.486,175.971,18.025,152.640
C00946=1092.880,116.806,-63.467,175.969,18.024,152.640
C00947=1092.876,116.557,-63.449,175.966,18.023,152.641
C00948=1092.870,116.307,-63.430,175.964,18.022,152.641
C00949=1092.864,116.058,-63.411,175.961,18.021,152.641
C00950=1092.859,115.809,-63.392,175.959,18.020,152.641
C00951=1092.853,115.560,-63.372,175.957,18.019,152.642
C00952=1092.848,115.310,-63.353,175.954,18.018,152.642
C00953=1092.843,115.061,-63.334,175.951,18.016,152.642
C00954=1092.836,114.812,-63.316,175.950,18.016,152.642
C00955=1092.831,114.563,-63.296,175.947,18.015,152.643
C00956=1092.825,114.314,-63.278,175.944,18.013,152.643
C00957=1092.820,114.065,-63.258,175.942,18.013,152.643
C00958=1092.814,113.815,-63.239,175.939,18.012,152.643
C00959=1092.808,113.566,-63.221,175.937,18.010,152.644
C00960=1092.803,113.317,-63.202,175.935,18.010,152.644
C00961=1092.797,113.067,-63.183,175.932,18.009,152.644
C00962=1092.792,112.818,-63.164,175.929,18.008,152.644
C00963=1092.786,112.570,-63.146,175.928,18.006,152.645
C00964=1092.780,112.320,-63.126,175.925,18.005,152.645
C00965=1092.774,112.044,-63.106,175.922,18.004,152.645
C00966=1092.768,111.767,-63.085,175.919,18.003,152.645
C00967=1092.761,111.491,-63.064,175.917,18.002,152.646
C00968=1092.755,111.215,-63.044,175.914,18.001,152.646
C00969=1092.750,110.965,-63.024,175.912,18.000,152.646
C00970=1092.744,110.717,-63.006,175.909,17.999,152.646
C00971=1092.738,110.467,-62.987,175.907,17.998,152.647
C00972=1092.733,110.217,-62.968,175.905,17.997,152.647
C00973=1092.727,109.969,-62.950,175.902,17.996,152.647
C00974=1092.721,109.719,-62.931,175.899,17.995,152.647
C00975=1092.716,109.470,-62.912,175.898,17.994,152.648
C00976=1092.710,109.221,-62.894,175.895,17.993,152.648
C00977=1092.704,108.971,-62.875,175.893,17.992,152.648
C00978=1092.698,108.723,-62.856,175.890,17.991,152.648
C00979=1092.693,108.473,-62.838,175.887,17.990,152.649
C00980=1092.687,108.224,-62.819,175.886,17.989,152.649
C00981=1092.682,107.975,-62.800,175.883,17.987,152.649
C00982=1092.676,107.725,-62.782,175.880,17.986,152.649
C00983=1092.670,107.477,-62.764,175.878,17.986,152.649
C00984=1092.665,107.227,-62.744,175.876,17.984,152.650
C00985=1092.659,106.977,-62.726,175.873,17.983,152.650
C00986=1092.654,106.729,-62.708,175.871,17.982,152.650
C00987=1092.648,106.479,-62.689,175.869,17.981,152.650
C00988=1092.642,106.230,-62.671,175.867,17.980,152.651
C00989=1092.637,105.981,-62.651,175.864,17.979,152.651
C00990=1092.630,105.731,-62.634,175.861,17.978,152.651
C00991=1092.625,105.482,-62.615,175.860,17.977,152.651
C00992=1092.619,105.233,-62.597,175.857,17.976,152.652
C00993=1092.614,104.984,-62.578,175.854,17.974,152.652
C00994=1092.608,104.734,-62.560,175.852,17.974,152.652
C00995=1092.603,104.485,-62.541,175.850,17.972,152.652
C00996=1092.597,104.236,-62.523,175.848,17.972,152.652
C00997=1092.592,103.987,-62.504,175.845,17.970,152.653
C00998=1092.586,103.737,-62.486,175.843,17.969,152.653
C00999=1092.581,103.488,-62.467,175.841,17.968,152.653
C01000=1092.574,103.239,-62.450,175.838,17.967,152.653
C01001=1092.569,102.990,-62.431,175.835,17.966,152.653
C01002=1092.563,102.740,-62.413,175.834,17.965,152.654
C01003=1092.558,102.492,-62.394,175.831,17.963,152.654
C01004=1092.552,102.242,-62.376,175.829,17.963,152.654
C01005=1092.547,101.992,-62.358,175.827,17.961,152.654
C01006=1092.541,101.743,-62.339,175.824,17.960,152.654
C01007=1092.536,101.494,-62.321,175.822,17.959,152.655
C01008=1092.530,101.245,-62.302,175.820,17.958,152.655
C01009=1092.525,100.995,-62.284,175.817,17.957,152.655
C01010=1092.518,100.746,-62.265,175.815,17.956,152.655
C01011=1092.513,100.497,-62.248,175.812,17.954,152.655
C01012=1092.508,100.247,-62.229,175.811,17.954,152.656
C01013=1092.502,99.999,-62.211,175.808,17.953,152.656
C01014=1092.496,99.749,-62.193,175.805,17.951,152.656
C01015=1092.491,99.500,-62.175,175.803,17.950,152.656
C01016=1092.484,99.251,-62.156,175.801,17.949,152.657
C01017=1092.479,99.002,-62.139,175.799,17.948,152.657
C01018=1092.473,98.752,-62.120,175.796,17.947,152.657
C01019=1092.468,98.503,-62.102,175.794,17.946,152.657
C01020=1092.462,98.253,-62.084,175.792,17.945,152.657
C01021=1092.457,98.004,-62.066,175.789,17.944,152.658
C01022=1092.451,97.754,-62.048,175.788,17.942,152.658
C01023=1092.445,97.506,-62.030,175.785,17.941,152.658
C01024=1092.439,97.257,-62.012,175.782,17.940,152.658
C01025=1092.434,97.007,-61.994,175.780,17.939,152.658
C01026=1092.428,96.758,-61.976,175.778,17.938,152.659
C01027=1092.422,96.509,-61.957,175.776,17.937,152.659
C01028=1092.416,96.260,-61.940,175.773,17.936,152.659
C01029=1092.410,95.983,-61.919,175.771,17.934,152.659
C01030=1092.404,95.707,-61.899,175.768,17.933,152.659
C01031=1092.398,95.431,-61.879,175.765,17.932,152.660
C01032=1092.391,95.154,-61.860,175.764,17.931,152.660
C01033=1092.386,94.905,-61.841,175.761,17.929,152.660
C01034=1092.380,94.656,-61.823,175.759,17.928,152.660
C01035=1092.375,94.407,-61.806,175.757,17.927,152.660
C01036=1092.369,94.158,-61.788,175.754,17.926,152.661
C01037=1092.364,93.907,-61.770,175.752,17.925,152.661
C01038=1092.358,93.658,-61.752,175.750,17.923,152.661
C01039=1092.352,93.409,-61.734,175.747,17.922,152.661
C01040=1092.346,93.160,-61.716,175.745,17.921,152.661
C01041=1092.341,92.911,-61.698,175.743,17.919,152.661
C01042=1092.335,92.661,-61.680,175.741,17.919,152.662
C01043=1092.330,92.412,-61.662,175.739,17.917,152.662
C01044=1092.324,92.163,-61.645,175.737,17.917,152.662
C01045=1092.318,91.913,-61.627,175.734,17.915,152.662
C01046=1092.313,91.664,-61.609,175.731,17.914,152.662
C01047=1092.308,91.415,-61.591,175.730,17.913,152.662
C01048=1092.302,91.165,-61.573,175.727,17.911,152.663
C01049=1092.296,90.916,-61.555,175.725,17.910,152.663
C01050=1092.291,90.667,-61.538,175.723,17.909,152.663
C01051=1092.285,90.417,-61.520,175.721,17.908,152.663
C01052=1092.279,90.168,-61.502,175.719,17.907,152.663
C01053=1092.274,89.919,-61.485,175.716,17.905,152.664
C01054=1092.268,89.670,-61.467,175.714,17.904,152.664
C01055=1092.262,89.421,-61.449,175.711,17.903,152.664
C01056=1092.256,89.171,-61.431,175.710,17.902,152.664
C01057=1092.250,88.922,-61.414,175.707,17.901,152.664
C01058=1092.245,88.673,-61.396,175.705,17.900,152.664
C01059=1092.239,88.423,-61.378,175.703,17.899,152.665
C01060=1092.233,88.174,-61.361,175.700,17.897,152.665
C01061=1092.228,87.925,-61.343,175.699,17.896,152.665
C01062=1092.222,87.675,-61.325,175.696,17.895,152.665
C01063=1092.216,87.426,-61.308,175.694,17.894,152.665
C01064=1092.211,87.176,-61.291,175.691,17.893,152.666
C01065=1092.205,86.927,-61.273,175.690,17.891,152.666
C01066=1092.199,86.678,-61.255,175.687,17.890,152.666
C01067=1092.194,86.429,-61.238,175.685,17.889,152.666
C01068=1092.188,86.180,-61.220,175.683,17.888,152.666
C01069=1092.182,85.930,-61.202,175.681,17.886,152.666
C01070=1092.177,85.681,-61.185,175.679,17.885,152.667
C01071=1092.171,85.431,-61.168,175.676,17.884,152.667
C01072=1092.166,85.182,-61.150,175.674,17.883,152.667
C01073=1092.160,84.932,-61.132,175.672,17.881,152.667
C01074=1092.154,84.683,-61.115,175.670,17.880,152.667
C01075=1092.149,84.434,-61.097,175.668,17.879,152.667
C01076=1092.144,84.185,-61.080,175.665,17.878,152.668
C01077=1092.137,83.935,-61.063,175.663,17.876,152.668
C01078=1092.131,83.686,-61.045,175.661,17.875,152.668
C01079=1092.126,83.437,-61.028,175.659,17.874,152.668
C01080=1092.120,83.188,-61.010,175.656,17.873,152.668
C01081=1092.114,82.938,-60.993,175.655,17.871,152.668
C01082=1092.109,82.689,-60.976,175.652,17.870,152.668
C01083=1092.103,82.440,-60.958,175.650,17.869,152.669
C01084=1092.098,82.190,-60.941,175.648,17.868,152.669
C01085=1092.093,81.941,-60.924,175.646,17.866,152.669
C01086=1092.086,81.691,-60.906,175.644,17.865,152.669
C01087=1092.081,81.442,-60.888,175.641,17.864,152.669
C01088=1092.075,81.193,-60.872,175.639,17.863,152.669
C01089=1092.069,80.944,-60.854,175.637,17.861,152.669
C01090=1092.064,80.695,-60.837,175.635,17.860,152.670
C01091=1092.058,80.444,-60.819,175.633,17.859,152.670
C01092=1092.053,80.195,-60.802,175.631,17.858,152.670
C01093=1092.047,79.919,-60.783,175.628,17.856,152.670
C01094=1092.041,79.643,-60.764,175.626,17.854,152.670
C01095=1092.034,79.367,-60.744,175.624,17.853,152.670
C01096=1092.028,79.091,-60.726,175.621,17.852,152.671
C01097=1092.022,78.842,-60.708,175.619,17.850,152.671
C01098=1092.017,78.592,-60.691,175.617,17.849,152.671
C01099=1092.011,78.343,-60.674,175.615,17.848,152.671
C01100=1092.005,78.093,-60.657,175.613,17.846,152.671
C01101=1092.000,77.844,-60.639,175.611,17.845,152.671
C01102=1091.994,77.594,-60.623,175.608,17.844,152.671
C01103=1091.988,77.345,-60.606,175.607,17.843,152.671
C01104=1091.983,77.096,-60.588,175.604,17.841,152.672
C01105=1091.977,76.847,-60.571,175.602,17.841,152.672
C01106=1091.971,76.597,-60.554,175.600,17.839,152.672
C01107=1091.965,76.348,-60.537,175.598,17.838,152.672
C01108=1091.960,76.099,-60.519,175.596,17.836,152.672
C01109=1091.954,75.849,-60.503,175.594,17.835,152.672
C01110=1091.948,75.600,-60.486,175.591,17.833,152.672
C01111=1091.943,75.351,-60.469,175.590,17.833,152.673
C01112=1091.937,75.102,-60.452,175.587,17.831,152.673
C01113=1091.931,74.851,-60.435,175.585,17.830,152.673
C01114=1091.926,74.602,-60.418,175.583,17.828,152.673
C01115=1091.920,74.353,-60.401,175.581,17.827,152.673
C01116=1091.914,74.103,-60.384,175.579,17.826,152.673
C01117=1091.909,73.854,-60.366,175.576,17.824,152.673
C01118=1091.903,73.605,-60.350,175.574,17.823,152.674
C01119=1091.897,73.356,-60.332,175.572,17.822,152.674
C01120=1091.892,73.106,-60.316,175.570,17.821,152.674
C01121=1091.886,72.857,-60.299,175.568,17.819,152.674
C01122=1091.881,72.608,-60.282,175.566,17.818,152.674
C01123=1091.875,72.359,-60.266,175.564,17.816,152.674
C01124=1091.869,72.109,-60.248,175.562,17.815,152.674
C01125=1091.863,71.859,-60.231,175.560,17.814,152.674
C01126=1091.857,71.610,-60.215,175.558,17.813,152.675
C01127=1091.852,71.361,-60.197,175.556,17.811,152.675
C01128=1091.846,71.111,-60.181,175.554,17.810,152.675
C01129=1091.841,70.862,-60.164,175.551,17.809,152.675
C01130=1091.835,70.613,-60.146,175.550,17.808,152.675
C01131=1091.829,70.363,-60.130,175.547,17.806,152.675
C01132=1091.824,70.114,-60.113,175.545,17.805,152.675
C01133=1091.818,69.864,-60.097,175.543,17.803,152.675
C01134=1091.813,69.615,-60.079,175.541,17.802,152.676
C01135=1091.807,69.366,-60.063,175.539,17.800,152.676
C01136=1091.801,69.116,-60.046,175.537,17.799,152.676
C01137=1091.796,68.867,-60.030,175.535,17.798,152.676
C01138=1091.790,68.618,-60.012,175.533,17.797,152.676
C01139=1091.784,68.369,-59.996,175.531,17.795,152.676
C01140=1091.779,68.119,-59.979,175.529,17.794,152.676
C01141=1091.773,67.870,-59.963,175.526,17.792,152.676
C01142=1091.767,67.621,-59.945,175.525,17.791,152.676
C01143=1091.761,67.371,-59.929,175.522,17.789,152.677
C01144=1091.755,67.122,-59.913,175.521,17.788,152.677
C01145=1091.750,66.872,-59.896,175.518,17.787,152.677
C01146=1091.744,66.623,-59.880,175.517,17.786,152.677
C01147=1091.739,66.374,-59.862,175.514,17.784,152.677
C01148=1091.733,66.124,-59.846,175.513,17.783,152.677
C01149=1091.728,65.875,-59.829,175.510,17.781,152.677
C01150=1091.722,65.625,-59.813,175.508,17.780,152.677
C01151=1091.716,65.376,-59.797,175.506,17.779,152.677
C01152=1091.711,65.126,-59.780,175.504,17.777,152.678
C01153=1091.705,64.877,-59.764,175.502,17.776,152.678
C01154=1091.699,64.627,-59.747,175.500,17.775,152.678
C01155=1091.693,64.379,-59.730,175.498,17.773,152.678
C01156=1091.687,64.129,-59.713,175.496,17.772,152.678
C01157=1091.680,63.852,-59.696,175.494,17.770,152.678
C01158=1091.674,63.576,-59.677,175.491,17.769,152.678
C01159=1091.668,63.300,-59.659,175.489,17.768,152.678
C01160=1091.661,63.024,-59.641,175.487,17.766,152.679
C01161=1091.656,62.774,-59.624,175.485,17.765,152.679
C01162=1091.650,62.525,-59.608,175.483,17.764,152.679
C01163=1091.644,62.276,-59.591,175.481,17.763,152.679
C01164=1091.638,62.027,-59.575,175.479,17.761,152.679
C01165=1091.633,61.777,-59.558,175.477,17.760,152.679
C01166=1091.627,61.528,-59.542,175.474,17.758,152.679
C01167=1091.621,61.278,-59.525,175.473,17.757,152.679
C01168=1091.615,61.029,-59.509,175.470,17.756,152.680
C01169=1091.609,60.780,-59.493,175.469,17.754,152.680
C01170=1091.604,60.530,-59.476,175.466,17.752,152.680
C01171=1091.598,60.281,-59.460,175.465,17.751,152.680
C01172=1091.592,60.031,-59.444,175.462,17.750,152.680
C01173=1091.586,59.781,-59.428,175.461,17.748,152.680
C01174=1091.580,59.532,-59.412,175.458,17.747,152.680
C01175=1091.574,59.283,-59.395,175.457,17.746,152.680
C01176=1091.569,59.033,-59.379,175.454,17.744,152.680
C01177=1091.563,58.784,-59.362,175.452,17.743,152.680
C01178=1091.558,58.535,-59.346,175.451,17.742,152.681
C01179=1091.552,58.286,-59.330,175.448,17.740,152.681
C01180=1091.546,58.036,-59.314,175.447,17.739,152.681
C01181=1091.540,57.787,-59.298,175.444,17.738,152.681
C01182=1091.535,57.537,-59.281,175.443,17.736,152.681
C01183=1091.529,57.287,-59.265,175.440,17.735,152.681
C01184=1091.523,57.038,-59.249,175.439,17.733,152.681
C01185=1091.517,56.789,-59.233,175.436,17.732,152.681
C01186=1091.511,56.539,-59.217,175.435,17.730,152.681
C01187=1091.505,56.290,-59.200,175.432,17.729,152.681
C01188=1091.500,56.041,-59.184,175.431,17.728,152.682
C01189=1091.494,55.791,-59.169,175.429,17.727,152.682
C01190=1091.489,55.542,-59.152,175.426,17.725,152.682
C01191=1091.483,55.292,-59.136,175.425,17.723,152.682
C01192=1091.477,55.043,-59.119,175.423,17.722,152.682
C01193=1091.471,54.794,-59.103,175.421,17.721,152.682
C01194=1091.465,54.544,-59.088,175.419,17.719,152.682
C01195=1091.460,54.295,-59.072,175.417,17.718,152.682
C01196=1091.454,54.046,-59.056,175.414,17.716,152.682
C01197=1091.448,53.796,-59.039,175.413,17.715,152.682
C01198=1091.443,53.546,-59.024,175.411,17.713,152.682
C01199=1091.437,53.297,-59.007,175.409,17.712,152.682
C01200=1091.431,53.047,-58.991,175.407,17.711,152.683
C01201=1091.426,52.798,-58.975,175.405,17.709,152.683
C01202=1091.420,52.549,-58.959,175.403,17.708,152.683
C01203=1091.414,52.299,-58.943,175.401,17.706,152.683
C01204=1091.408,52.050,-58.927,175.399,17.705,152.683
C01205=1091.403,51.800,-58.911,175.397,17.703,152.683
C01206=1091.397,51.551,-58.895,175.395,17.702,152.683
C01207=1091.392,51.302,-58.879,175.393,17.700,152.683
C01208=1091.386,51.052,-58.863,175.391,17.699,152.683
C01209=1091.380,50.803,-58.847,175.390,17.698,152.683
C01210=1091.375,50.553,-58.832,175.387,17.696,152.683
C01211=1091.369,50.304,-58.816,175.386,17.695,152.683
C01212=1091.363,50.055,-58.800,175.383,17.693,152.683
C01213=1091.357,49.805,-58.784,175.382,17.692,152.684
C01214=1091.352,49.556,-58.768,175.379,17.690,152.684
C01215=1091.346,49.306,-58.753,175.378,17.689,152.684
C01216=1091.340,49.057,-58.736,175.375,17.687,152.684
C01217=1091.334,48.807,-58.720,175.374,17.686,152.684
C01218=1091.329,48.558,-58.705,175.372,17.684,152.684
C01219=1091.323,48.309,-58.689,175.370,17.683,152.684
C01220=1091.318,48.059,-58.673,175.368,17.682,152.684
C01221=1091.312,47.782,-58.655,175.366,17.679,152.684
C01222=1091.306,47.506,-58.637,175.364,17.678,152.684
C01223=1091.299,47.229,-58.620,175.362,17.677,152.684
C01224=1091.293,46.953,-58.602,175.360,17.675,152.684
C01225=1091.288,46.704,-58.587,175.358,17.674,152.684
C01226=1091.282,46.454,-58.571,175.356,17.672,152.685
C01227=1091.276,46.205,-58.555,175.354,17.670,152.684
C01228=1091.271,45.955,-58.540,175.352,17.669,152.685
C01229=1091.265,45.706,-58.523,175.350,17.668,152.685
C01230=1091.260,45.456,-58.508,175.348,17.665,152.685
C01231=1091.254,45.207,-58.493,175.346,17.664,152.685
C01232=1091.249,44.958,-58.476,175.345,17.663,152.685
C01233=1091.243,44.708,-58.461,175.343,17.661,152.685
C01234=1091.238,44.459,-58.445,175.341,17.660,152.685
C01235=1091.232,44.209,-58.429,175.339,17.658,152.685
C01236=1091.226,43.960,-58.413,175.337,17.657,152.685
C01237=1091.220,43.711,-58.399,175.335,17.655,152.685
C01238=1091.215,43.461,-58.383,175.333,17.654,152.685
C01239=1091.209,43.211,-58.367,175.332,17.652,152.685
C01240=1091.204,42.962,-58.352,175.329,17.651,152.685
C01241=1091.198,42.713,-58.335,175.328,17.649,152.685
C01242=1091.191,42.463,-58.320,175.325,17.648,152.685
C01243=1091.186,42.214,-58.305,175.324,17.646,152.686
C01244=1091.180,41.964,-58.289,175.322,17.645,152.685
C01245=1091.175,41.714,-58.273,175.320,17.643,152.686
C01246=1091.170,41.465,-58.258,175.318,17.642,152.686
C01247=1091.163,41.216,-58.243,175.316,17.640,152.686
C01248=1091.157,40.966,-58.227,175.314,17.639,152.686
C01249=1091.152,40.717,-58.212,175.313,17.638,152.686
C01250=1091.146,40.468,-58.196,175.311,17.636,152.686
C01251=1091.140,40.218,-58.181,175.309,17.635,152.686
C01252=1091.135,39.969,-58.165,175.306,17.633,152.686
C01253=1091.129,39.719,-58.150,175.305,17.631,152.686
C01254=1091.124,39.470,-58.134,175.303,17.630,152.686
C01255=1091.117,39.220,-58.119,175.301,17.628,152.686
C01256=1091.112,38.970,-58.104,175.300,17.627,152.686
C01257=1091.107,38.721,-58.088,175.297,17.625,152.686
C01258=1091.101,38.472,-58.072,175.296,17.624,152.686
C01259=1091.095,38.223,-58.058,175.293,17.622,152.686
C01260=1091.089,37.973,-58.042,175.292,17.621,152.686
C01261=1091.084,37.723,-58.026,175.290,17.619,152.686
C01262=1091.078,37.475,-58.011,175.288,17.618,152.687
C01263=1091.072,37.225,-57.996,175.286,17.616,152.687
C01264=1091.066,36.975,-57.980,175.285,17.615,152.687
C01265=1091.061,36.726,-57.966,175.282,17.613,152.687
C01266=1091.055,36.476,-57.950,175.281,17.612,152.687
C01267=1091.049,36.227,-57.935,175.278,17.610,152.687
C01268=1091.043,35.977,-57.919,175.277,17.609,152.687
C01269=1091.037,35.728,-57.904,175.275,17.608,152.687
C01270=1091.032,35.478,-57.889,175.273,17.606,152.687
C01271=1091.026,35.229,-57.873,175.272,17.604,152.687
C01272=1091.020,34.980,-57.859,175.269,17.603,152.687
C01273=1091.015,34.730,-57.843,175.268,17.602,152.687
C01274=1091.008,34.480,-57.828,175.266,17.600,152.687
C01275=1091.003,34.231,-57.813,175.264,17.598,152.687
C01276=1090.997,33.982,-57.798,175.262,17.597,152.687
C01277=1090.991,33.732,-57.782,175.261,17.596,152.687
C01278=1090.985,33.483,-57.767,175.258,17.594,152.688
C01279=1090.980,33.233,-57.752,175.257,17.592,152.687
C01280=1090.974,32.983,-57.737,175.254,17.591,152.688
C01281=1090.968,32.734,-57.722,175.253,17.589,152.688
C01282=1090.963,32.485,-57.707,175.251,17.588,152.688
C01283=1090.957,32.235,-57.692,175.249,17.586,152.688
C01284=1090.952,31.986,-57.676,175.248,17.585,152.688
C01285=1090.944,31.709,-57.660,175.245,17.583,152.688
C01286=1090.938,31.432,-57.643,175.244,17.582,152.688
C01287=1090.932,31.156,-57.627,175.241,17.579,152.688
C01288=1090.926,30.880,-57.609,175.239,17.578,152.688
C01289=1090.920,30.631,-57.595,175.238,17.576,152.688
C01290=1090.914,30.381,-57.579,175.236,17.575,152.688
C01291=1090.909,30.132,-57.565,175.234,17.574,152.688
C01292=1090.903,29.882,-57.549,175.232,17.572,152.688
C01293=1090.897,29.633,-57.535,175.231,17.571,152.688
C01294=1090.892,29.383,-57.519,175.228,17.569,152.688
C01295=1090.886,29.134,-57.505,175.227,17.568,152.688
C01296=1090.880,28.884,-57.489,175.225,17.565,152.688
C01297=1090.875,28.635,-57.475,175.223,17.564,152.688
C01298=1090.869,28.385,-57.460,175.222,17.563,152.688
C01299=1090.863,28.136,-57.445,175.219,17.561,152.688
C01300=1090.857,27.886,-57.430,175.218,17.560,152.688
C01301=1090.852,27.637,-57.415,175.216,17.558,152.688
C01302=1090.845,27.387,-57.400,175.214,17.556,152.688
C01303=1090.840,27.138,-57.385,175.212,17.555,152.689
C01304=1090.834,26.888,-57.370,175.211,17.554,152.688
C01305=1090.828,26.639,-57.355,175.208,17.552,152.689
C01306=1090.823,26.389,-57.340,175.207,17.550,152.689
C01307=1090.817,26.140,-57.326,175.205,17.549,152.689
C01308=1090.811,25.890,-57.311,175.203,17.548,152.689
C01309=1090.806,25.641,-57.296,175.202,17.546,152.689
C01310=1090.799,25.391,-57.281,175.199,17.544,152.689
C01311=1090.793,25.142,-57.266,175.198,17.543,152.689
C01312=1090.788,24.892,-57.251,175.196,17.542,152.689
C01313=1090.782,24.643,-57.237,175.194,17.540,152.689
C01314=1090.776,24.393,-57.222,175.192,17.538,152.689
C01315=1090.770,24.144,-57.207,175.191,17.537,152.689
C01316=1090.765,23.894,-57.192,175.188,17.535,152.689
C01317=1090.759,23.644,-57.178,175.187,17.534,152.689
C01318=1090.753,23.395,-57.163,175.185,17.533,152.689
C01319=1090.748,23.146,-57.148,175.183,17.530,152.689
C01320=1090.742,22.897,-57.133,175.182,17.529,152.689
C01321=1090.736,22.646,-57.119,175.180,17.528,152.689
C01322=1090.730,22.397,-57.104,175.178,17.526,152.689
C01323=1090.725,22.148,-57.089,175.176,17.524,152.689
C01324=1090.719,21.898,-57.075,175.175,17.523,152.689
C01325=1090.713,21.649,-57.060,175.173,17.521,152.689
C01326=1090.707,21.399,-57.045,175.171,17.520,152.689
C01327=1090.702,21.150,-57.030,175.170,17.519,152.689
C01328=1090.696,20.900,-57.016,175.167,17.516,152.689
C01329=1090.690,20.651,-57.001,175.166,17.515,152.690
C01330=1090.685,20.401,-56.986,175.164,17.514,152.689
C01331=1090.679,20.151,-56.972,175.162,17.512,152.690
C01332=1090.673,19.902,-56.957,175.160,17.510,152.690
C01333=1090.667,19.653,-56.943,175.159,17.509,152.690
C01334=1090.661,19.403,-56.929,175.157,17.507,152.690
C01335=1090.655,19.154,-56.914,175.155,17.506,152.690
C01336=1090.650,18.903,-56.899,175.154,17.505,152.690
C01337=1090.644,18.654,-56.885,175.151,17.503,152.690
C01338=1090.638,18.405,-56.870,175.150,17.501,152.690
C01339=1090.632,18.155,-56.856,175.148,17.500,152.690
C01340=1090.627,17.906,-56.841,175.146,17.498,152.690
C01341=1090.621,17.657,-56.827,175.145,17.496,152.690
C01342=1090.615,17.407,-56.812,175.143,17.495,152.690
C01343=1090.610,17.157,-56.798,175.141,17.493,152.690
C01344=1090.604,16.907,-56.783,175.139,17.492,152.690
C01345=1090.598,16.659,-56.768,175.138,17.491,152.690
C01346=1090.592,16.409,-56.755,175.135,17.489,152.690
C01347=1090.586,16.159,-56.740,175.134,17.487,152.690
C01348=1090.580,15.910,-56.726,175.133,17.486,152.690
C01349=1090.575,15.635,-56.710,175.130,17.484,152.690
C01350=1090.567,15.360,-56.694,175.129,17.482,152.690
C01351=1090.562,15.085,-56.678,175.126,17.481,152.690
C01352=1090.556,14.810,-56.662,175.125,17.479,152.690
C01353=1090.549,14.560,-56.647,175.123,17.477,152.690
C01354=1090.544,14.311,-56.633,175.121,17.476,152.690
C01355=1090.538,14.062,-56.619,175.120,17.474,152.690
C01356=1090.532,13.811,-56.604,175.117,17.473,152.690
C01357=1090.527,13.562,-56.591,175.116,17.471,152.690
C01358=1090.521,13.313,-56.576,175.114,17.470,152.690
C01359=1090.514,13.063,-56.562,175.112,17.468,152.690
C01360=1090.508,12.814,-56.548,175.110,17.467,152.690
C01361=1090.503,12.564,-56.534,175.109,17.465,152.690
C01362=1090.496,12.315,-56.519,175.107,17.464,152.691
C01363=1090.491,12.065,-56.505,175.105,17.462,152.691
C01364=1090.485,11.815,-56.491,175.104,17.461,152.691
C01365=1090.479,11.566,-56.476,175.102,17.459,152.691
C01366=1090.474,11.316,-56.462,175.100,17.457,152.691
C01367=1090.468,11.067,-56.448,175.098,17.456,152.691
C01368=1090.462,10.817,-56.434,175.097,17.454,152.691
C01369=1090.456,10.567,-56.420,175.095,17.453,152.691
C01370=1090.450,10.318,-56.405,175.093,17.451,152.691
C01371=1090.444,10.069,-56.392,175.092,17.450,152.691
C01372=1090.438,9.819,-56.378,175.090,17.449,152.691
C01373=1090.432,9.570,-56.363,175.088,17.447,152.691
C01374=1090.427,9.320,-56.349,175.086,17.445,152.691
C01375=1090.421,9.070,-56.335,175.085,17.444,152.691
C01376=1090.415,8.821,-56.320,175.083,17.442,152.691
C01377=1090.410,8.572,-56.307,175.081,17.440,152.691
C01378=1090.403,8.321,-56.292,175.080,17.439,152.691
C01379=1090.398,8.072,-56.278,175.078,17.438,152.691
C01380=1090.391,7.823,-56.264,175.076,17.436,152.691
C01381=1090.386,7.574,-56.251,175.074,17.434,152.691
C01382=1090.380,7.323,-56.236,175.073,17.433,152.691
C01383=1090.374,7.074,-56.222,175.071,17.431,152.691
C01384=1090.369,6.825,-56.208,175.069,17.430,152.691
C01385=1090.363,6.575,-56.194,175.068,17.429,152.691
C01386=1090.357,6.325,-56.180,175.066,17.427,152.691
C01387=1090.351,6.076,-56.166,175.064,17.425,152.691
C01388=1090.345,5.827,-56.152,175.062,17.424,152.691
C01389=1090.340,5.577,-56.138,175.061,17.422,152.691
C01390=1090.334,5.328,-56.124,175.058,17.420,152.691
C01391=1090.328,5.077,-56.110,175.057,17.419,152.691
C01392=1090.322,4.828,-56.095,175.056,17.417,152.691
C01393=1090.316,4.579,-56.082,175.054,17.416,152.691
C01394=1090.311,4.329,-56.068,175.052,17.414,152.691
C01395=1090.305,4.080,-56.054,175.050,17.413,152.691
C01396=1090.299,3.830,-56.040,175.049,17.411,152.691
C01397=1090.294,3.580,-56.026,175.047,17.409,152.691
C01398=1090.287,3.331,-56.012,175.045,17.408,152.691
C01399=1090.282,3.082,-55.999,175.044,17.407,152.691
C01400=1090.276,2.832,-55.985,175.042,17.405,152.691
C01401=1090.271,2.583,-55.971,175.040,17.403,152.691
C01402=1090.265,2.332,-55.957,175.039,17.402,152.691
C01403=1090.258,2.083,-55.943,175.037,17.400,152.691
C01404=1090.253,1.834,-55.929,175.036,17.399,152.691
C01405=1090.247,1.584,-55.916,175.033,17.397,152.691
C01406=1090.242,1.334,-55.902,175.032,17.396,152.692
C01407=1090.236,1.085,-55.888,175.030,17.394,152.692
C01408=1090.230,0.836,-55.875,175.028,17.392,152.692
C01409=1090.224,0.587,-55.860,175.027,17.391,152.692
C01410=1090.218,0.336,-55.846,175.025,17.389,152.692
C01411=1090.213,0.087,-55.832,175.024,17.388,152.691
C01412=1090.207,-0.163,-55.819,175.021,17.386,152.692
C01413=1090.201,-0.436,-55.804,175.020,17.384,152.692
C01414=1090.194,-0.709,-55.789,175.018,17.382,152.692
C01415=1090.188,-0.982,-55.773,175.016,17.381,152.692
C01416=1090.183,-1.255,-55.758,175.015,17.380,152.692
C01417=1090.176,-1.504,-55.745,175.013,17.377,152.692
C01418=1090.171,-1.754,-55.731,175.011,17.376,152.692
C01419=1090.166,-2.003,-55.717,175.010,17.375,152.692
C01420=1090.159,-2.253,-55.704,175.007,17.373,152.692
C01421=1090.153,-2.503,-55.690,175.006,17.371,152.692
C01422=1090.148,-2.752,-55.676,175.004,17.370,152.692
C01423=1090.142,-3.002,-55.662,175.003,17.368,152.692
C01424=1090.136,-3.251,-55.649,175.001,17.366,152.692
C01425=1090.131,-3.501,-55.635,174.999,17.365,152.692
C01426=1090.124,-3.750,-55.622,174.998,17.363,152.692
C01427=1090.119,-4.000,-55.608,174.996,17.362,152.692
C01428=1090.114,-4.250,-55.595,174.994,17.360,152.692
C01429=1090.108,-4.499,-55.581,174.993,17.359,152.692
C01430=1090.101,-4.749,-55.567,174.991,17.358,152.692
C01431=1090.095,-4.999,-55.554,174.990,17.356,152.692
C01432=1090.090,-5.248,-55.540,174.987,17.354,152.692
C01433=1090.084,-5.498,-55.527,174.986,17.353,152.692
C01434=1090.078,-5.747,-55.513,174.984,17.351,152.692
C01435=1090.072,-5.996,-55.500,174.983,17.350,152.692
C01436=1090.066,-6.246,-55.486,174.981,17.348,152.692
C01437=1090.060,-6.496,-55.473,174.979,17.347,152.692
C01438=1090.055,-6.745,-55.459,174.978,17.345,152.692
C01439=1090.049,-6.995,-55.446,174.976,17.344,152.692
C01440=1090.043,-7.244,-55.432,174.975,17.342,152.692
C01441=1090.037,-7.494,-55.419,174.972,17.340,152.692
C01442=1090.031,-7.744,-55.405,174.971,17.339,152.692
C01443=1090.025,-7.994,-55.392,174.969,17.338,152.692
C01444=1090.019,-8.243,-55.379,174.968,17.336,152.692
C01445=1090.013,-8.493,-55.365,174.966,17.334,152.692
C01446=1090.007,-8.742,-55.352,174.964,17.333,152.692
C01447=1090.002,-8.992,-55.339,174.963,17.331,152.692
C01448=1089.996,-9.241,-55.325,174.961,17.330,152.692
C01449=1089.990,-9.491,-55.312,174.960,17.328,152.692
C01450=1089.984,-9.740,-55.298,174.957,17.327,152.692
C01451=1089.979,-9.990,-55.285,174.956,17.325,152.692
C01452=1089.973,-10.240,-55.272,174.955,17.324,152.692
C01453=1089.967,-10.489,-55.258,174.953,17.323,152.692
C01454=1089.961,-10.738,-55.245,174.951,17.320,152.692
C01455=1089.955,-10.988,-55.232,174.950,17.319,152.692
C01456=1089.950,-11.238,-55.218,174.948,17.318,152.692
C01457=1089.943,-11.487,-55.205,174.947,17.316,152.692
C01458=1089.938,-11.737,-55.192,174.944,17.314,152.692
C01459=1089.932,-11.987,-55.179,174.943,17.313,152.692
C01460=1089.927,-12.236,-55.165,174.941,17.311,152.692
C01461=1089.921,-12.486,-55.152,174.940,17.310,152.692
C01462=1089.914,-12.735,-55.139,174.938,17.309,152.692
C01463=1089.909,-12.985,-55.125,174.936,17.306,152.692
C01464=1089.903,-13.235,-55.113,174.935,17.305,152.693
C01465=1089.898,-13.484,-55.099,174.933,17.304,152.692
C01466=1089.891,-13.734,-55.085,174.932,17.302,152.692
C01467=1089.885,-13.983,-55.073,174.930,17.301,152.692
C01468=1089.880,-14.233,-55.059,174.928,17.299,152.692
C01469=1089.874,-14.482,-55.046,174.927,17.297,152.692
C01470=1089.869,-14.732,-55.033,174.925,17.296,152.693
C01471=1089.863,-14.981,-55.020,174.924,17.295,152.692
C01472=1089.857,-15.231,-55.007,174.921,17.292,152.692
C01473=1089.852,-15.481,-54.993,174.920,17.291,152.693
C01474=1089.846,-15.730,-54.981,174.918,17.290,152.693
C01475=1089.839,-15.980,-54.967,174.917,17.289,152.693
C01476=1089.833,-16.229,-54.954,174.915,17.287,152.693
C01477=1089.827,-16.502,-54.940,174.913,17.285,152.693
C01478=1089.820,-16.773,-54.926,174.912,17.284,152.693
C01479=1089.815,-17.044,-54.911,174.910,17.282,152.693
C01480=1089.808,-17.315,-54.897,174.908,17.280,152.693
C01481=1089.802,-17.565,-54.885,174.906,17.279,152.693
C01482=1089.796,-17.814,-54.871,174.905,17.277,152.693
C01483=1089.790,-18.064,-54.858,174.903,17.276,152.693
C01484=1089.784,-18.314,-54.845,174.901,17.274,152.693
C01485=1089.778,-18.563,-54.832,174.900,17.272,152.693
C01486=1089.772,-18.813,-54.819,174.898,17.271,152.693
C01487=1089.766,-19.063,-54.807,174.897,17.270,152.693
C01488=1089.761,-19.312,-54.793,174.895,17.269,152.693
C01489=1089.755,-19.562,-54.780,174.893,17.266,152.693
C01490=1089.749,-19.811,-54.767,174.892,17.265,152.693
C01491=1089.743,-20.061,-54.755,174.890,17.264,152.693
C01492=1089.737,-20.310,-54.742,174.889,17.262,152.693
C01493=1089.731,-20.560,-54.729,174.887,17.261,152.693
C01494=1089.726,-20.809,-54.715,174.885,17.259,152.693
C01495=1089.720,-21.059,-54.703,174.884,17.257,152.693
C01496=1089.714,-21.309,-54.690,174.882,17.256,152.693
C01497=1089.708,-21.558,-54.677,174.881,17.255,152.693
C01498=1089.702,-21.808,-54.664,174.879,17.254,152.693
C01499=1089.696,-22.057,-54.651,174.878,17.252,152.693
C01500=1089.691,-22.307,-54.638,174.875,17.250,152.693
C01501=1089.685,-22.557,-54.626,174.874,17.249,152.693
C01502=1089.679,-22.806,-54.612,174.872,17.247,152.693
C01503=1089.673,-23.056,-54.600,174.871,17.246,152.693
C01504=1089.667,-23.305,-54.586,174.869,17.244,152.693
C01505=1089.661,-23.555,-54.574,174.867,17.242,152.693
C01506=1089.655,-23.805,-54.561,174.866,17.241,152.693
C01507=1089.650,-24.054,-54.548,174.864,17.240,152.693
C01508=1089.644,-24.304,-54.535,174.863,17.238,152.693
C01509=1089.638,-24.554,-54.523,174.861,17.237,152.693
C01510=1089.632,-24.803,-54.509,174.860,17.235,152.693
C01511=1089.626,-25.053,-54.497,174.857,17.234,152.693
C01512=1089.620,-25.303,-54.484,174.856,17.232,152.693
C01513=1089.615,-25.552,-54.472,174.855,17.230,152.693
C01514=1089.609,-25.801,-54.459,174.853,17.229,152.693
C01515=1089.604,-26.051,-54.446,174.852,17.228,152.693
C01516=1089.598,-26.301,-54.433,174.850,17.227,152.693
C01517=1089.592,-26.551,-54.421,174.848,17.224,152.693
C01518=1089.586,-26.800,-54.408,174.846,17.223,152.693
C01519=1089.580,-27.049,-54.395,174.845,17.222,152.694
C01520=1089.574,-27.299,-54.383,174.843,17.220,152.693
C01521=1089.569,-27.549,-54.370,174.842,17.219,152.694
C01522=1089.562,-27.799,-54.357,174.840,17.217,152.694
C01523=1089.556,-28.048,-54.344,174.838,17.216,152.694
C01524=1089.551,-28.298,-54.332,174.837,17.214,152.694
C01525=1089.544,-28.547,-54.320,174.835,17.213,152.694
C01526=1089.538,-28.796,-54.307,174.834,17.211,152.694
C01527=1089.532,-29.046,-54.294,174.832,17.210,152.694
C01528=1089.526,-29.296,-54.282,174.831,17.209,152.694
C01529=1089.521,-29.546,-54.269,174.829,17.207,152.694
C01530=1089.515,-29.795,-54.257,174.827,17.205,152.694
C01531=1089.509,-30.045,-54.244,174.826,17.204,152.694
C01532=1089.503,-30.294,-54.231,174.824,17.203,152.694
C01533=1089.497,-30.544,-54.219,174.823,17.201,152.694
C01534=1089.491,-30.794,-54.206,174.821,17.200,152.694
C01535=1089.486,-31.043,-54.194,174.820,17.198,152.694
C01536=1089.480,-31.293,-54.181,174.818,17.197,152.694
C01537=1089.473,-31.543,-54.169,174.816,17.195,152.694
C01538=1089.468,-31.793,-54.157,174.814,17.194,152.694
C01539=1089.462,-32.041,-54.144,174.813,17.193,152.694
C01540=1089.456,-32.291,-54.131,174.811,17.191,152.694
C01541=1089.449,-32.562,-54.117,174.810,17.190,152.694
C01542=1089.444,-32.833,-54.104,174.808,17.188,152.694
C01543=1089.437,-33.103,-54.091,174.806,17.186,152.694
C01544=1089.430,-33.374,-54.077,174.805,17.185,152.694
C01545=1089.425,-33.623,-54.065,174.803,17.183,152.694
C01546=1089.419,-33.873,-54.053,174.801,17.182,152.694
C01547=1089.413,-34.123,-54.040,174.799,17.180,152.694
C01548=1089.407,-34.373,-54.028,174.798,17.179,152.694
C01549=1089.401,-34.622,-54.016,174.796,17.177,152.694
C01550=1089.395,-34.872,-54.003,174.795,17.176,152.694
C01551=1089.389,-35.122,-53.991,174.793,17.175,152.694
C01552=1089.384,-35.371,-53.979,174.792,17.173,152.694
C01553=1089.378,-35.621,-53.966,174.790,17.172,152.694
C01554=1089.372,-35.870,-53.954,174.788,17.170,152.694
C01555=1089.366,-36.120,-53.941,174.787,17.169,152.694
C01556=1089.360,-36.369,-53.929,174.785,17.167,152.694
C01557=1089.354,-36.619,-53.917,174.784,17.166,152.694
C01558=1089.348,-36.869,-53.904,174.782,17.164,152.695
C01559=1089.343,-37.118,-53.892,174.781,17.163,152.694
C01560=1089.337,-37.368,-53.880,174.779,17.162,152.695
C01561=1089.331,-37.618,-53.868,174.778,17.160,152.695
C01562=1089.325,-37.867,-53.855,174.775,17.158,152.695
C01563=1089.319,-38.117,-53.843,174.774,17.157,152.695
C01564=1089.313,-38.367,-53.830,174.772,17.156,152.695
C01565=1089.308,-38.616,-53.818,174.771,17.154,152.695
C01566=1089.302,-38.865,-53.806,174.769,17.153,152.695
C01567=1089.296,-39.115,-53.794,174.768,17.151,152.695
C01568=1089.290,-39.364,-53.781,174.766,17.150,152.695
C01569=1089.284,-39.615,-53.770,174.765,17.149,152.695
C01570=1089.278,-39.864,-53.758,174.763,17.148,152.695
C01571=1089.272,-40.114,-53.745,174.761,17.146,152.695
C01572=1089.266,-40.363,-53.733,174.760,17.144,152.695
C01573=1089.260,-40.613,-53.721,174.758,17.143,152.695
C01574=1089.254,-40.863,-53.708,174.757,17.142,152.695
C01575=1089.248,-41.112,-53.697,174.755,17.140,152.695
C01576=1089.242,-41.362,-53.684,174.754,17.139,152.695
C01577=1089.237,-41.612,-53.672,174.752,17.137,152.695
C01578=1089.231,-41.861,-53.661,174.751,17.136,152.695
C01579=1089.225,-42.111,-53.648,174.749,17.135,152.695
C01580=1089.218,-42.361,-53.636,174.748,17.134,152.695
C01581=1089.213,-42.610,-53.624,174.746,17.132,152.695
C01582=1089.207,-42.860,-53.612,174.744,17.130,152.695
C01583=1089.201,-43.110,-53.600,174.742,17.129,152.695
C01584=1089.195,-43.359,-53.588,174.741,17.128,152.695
C01585=1089.189,-43.609,-53.576,174.739,17.126,152.695
C01586=1089.183,-43.858,-53.564,174.738,17.125,152.695
C01587=1089.177,-44.108,-53.551,174.736,17.123,152.695
C01588=1089.171,-44.358,-53.540,174.735,17.122,152.696
C01589=1089.166,-44.607,-53.528,174.733,17.121,152.696
C01590=1089.160,-44.857,-53.515,174.732,17.120,152.696
C01591=1089.153,-45.106,-53.503,174.730,17.118,152.696
C01592=1089.148,-45.356,-53.492,174.729,17.117,152.696
C01593=1089.142,-45.606,-53.480,174.726,17.115,152.696
C01594=1089.136,-45.856,-53.467,174.725,17.114,152.696
C01595=1089.130,-46.105,-53.457,174.723,17.112,152.696
C01596=1089.124,-46.355,-53.444,174.722,17.111,152.696
C01597=1089.119,-46.604,-53.432,174.720,17.110,152.696
C01598=1089.112,-46.854,-53.420,174.719,17.108,152.696
C01599=1089.107,-47.104,-53.408,174.717,17.107,152.696
C01600=1089.100,-47.353,-53.396,174.716,17.105,152.696
C01601=1089.094,-47.603,-53.384,174.714,17.104,152.696
C01602=1089.089,-47.853,-53.373,174.713,17.103,152.696
C01603=1089.083,-48.103,-53.360,174.711,17.102,152.696
C01604=1089.078,-48.352,-53.348,174.710,17.100,152.696
C01605=1089.070,-48.623,-53.336,174.708,17.098,152.696
C01606=1089.065,-48.894,-53.323,174.706,17.097,152.696
C01607=1089.058,-49.165,-53.310,174.705,17.096,152.696
C01608=1089.052,-49.436,-53.297,174.703,17.094,152.696
C01609=1089.046,-49.685,-53.285,174.702,17.093,152.696
C01610=1089.040,-49.936,-53.274,174.700,17.092,152.696
C01611=1089.034,-50.184,-53.262,174.698,17.090,152.696
C01612=1089.028,-50.434,-53.249,174.696,17.089,152.697
C01613=1089.023,-50.684,-53.239,174.695,17.087,152.696
C01614=1089.016,-50.933,-53.227,174.693,17.086,152.697
C01615=1089.010,-51.184,-53.215,174.692,17.085,152.697
C01616=1089.004,-51.433,-53.203,174.690,17.083,152.697
C01617=1088.998,-51.682,-53.191,174.689,17.082,152.697
C01618=1088.992,-51.933,-53.179,174.687,17.081,152.697
C01619=1088.986,-52.182,-53.168,174.686,17.079,152.697
C01620=1088.980,-52.432,-53.157,174.684,17.078,152.697
C01621=1088.974,-52.681,-53.145,174.682,17.077,152.697
C01622=1088.968,-52.931,-53.133,174.681,17.076,152.697
C01623=1088.961,-53.181,-53.121,174.679,17.074,152.697
C01624=1088.956,-53.430,-53.110,174.678,17.073,152.697
C01625=1088.950,-53.680,-53.098,174.676,17.072,152.697
C01626=1088.944,-53.929,-53.086,174.675,17.071,152.697
C01627=1088.937,-54.179,-53.075,174.673,17.070,152.697
C01628=1088.931,-54.428,-53.063,174.672,17.068,152.697
C01629=1088.926,-54.679,-53.051,174.670,17.067,152.697
C01630=1088.920,-54.927,-53.040,174.668,17.066,152.698
C01631=1088.913,-55.178,-53.029,174.667,17.064,152.697
C01632=1088.907,-55.428,-53.017,174.665,17.063,152.698
C01633=1088.902,-55.677,-53.005,174.664,17.062,152.698
C01634=1088.895,-55.927,-52.994,174.662,17.060,152.698
C01635=1088.889,-56.176,-52.982,174.661,17.059,152.698
C01636=1088.883,-56.426,-52.971,174.658,17.058,152.698
C01637=1088.878,-56.676,-52.959,174.657,17.056,152.698
C01638=1088.871,-56.926,-52.948,174.655,17.055,152.698
C01639=1088.865,-57.175,-52.936,174.654,17.054,152.698
C01640=1088.859,-57.425,-52.925,174.652,17.052,152.698
C01641=1088.854,-57.675,-52.913,174.651,17.051,152.698
C01642=1088.847,-57.924,-52.901,174.649,17.050,152.698
C01643=1088.842,-58.174,-52.891,174.648,17.048,152.698
C01644=1088.835,-58.423,-52.879,174.646,17.047,152.698
C01645=1088.829,-58.673,-52.868,174.644,17.046,152.698
C01646=1088.824,-58.923,-52.856,174.643,17.045,152.698
C01647=1088.818,-59.172,-52.844,174.641,17.043,152.699
C01648=1088.811,-59.422,-52.833,174.640,17.042,152.699
C01649=1088.805,-59.672,-52.822,174.638,17.041,152.699
C01650=1088.799,-59.921,-52.810,174.637,17.040,152.699
C01651=1088.794,-60.171,-52.799,174.635,17.039,152.699
C01652=1088.787,-60.421,-52.787,174.634,17.037,152.699
C01653=1088.781,-60.670,-52.776,174.632,17.036,152.699
C01654=1088.775,-60.920,-52.765,174.631,17.035,152.699
C01655=1088.769,-61.170,-52.754,174.629,17.034,152.699
C01656=1088.764,-61.419,-52.742,174.628,17.032,152.699
C01657=1088.758,-61.669,-52.730,174.626,17.031,152.699
C01658=1088.752,-61.919,-52.719,174.624,17.030,152.699
C01659=1088.745,-62.168,-52.708,174.623,17.028,152.699
C01660=1088.740,-62.418,-52.697,174.621,17.027,152.699
C01661=1088.734,-62.668,-52.685,174.620,17.026,152.699
C01662=1088.728,-62.917,-52.673,174.618,17.025,152.700
C01663=1088.722,-63.167,-52.662,174.617,17.023,152.699
C01664=1088.716,-63.417,-52.651,174.615,17.022,152.700
C01665=1088.710,-63.666,-52.640,174.613,17.021,152.700
C01666=1088.703,-63.916,-52.628,174.612,17.020,152.700
C01667=1088.698,-64.165,-52.617,174.610,17.018,152.700
C01668=1088.693,-64.415,-52.606,174.609,17.017,152.700
C01669=1088.685,-64.688,-52.594,174.607,17.016,152.700
C01670=1088.679,-64.960,-52.581,174.606,17.015,152.700
C01671=1088.673,-65.232,-52.569,174.604,17.014,152.700
C01672=1088.666,-65.504,-52.557,174.603,17.012,152.700
C01673=1088.661,-65.754,-52.546,174.601,17.011,152.700
C01674=1088.654,-66.004,-52.534,174.600,17.010,152.700
C01675=1088.649,-66.254,-52.523,174.598,17.009,152.700
C01676=1088.643,-66.503,-52.513,174.596,17.008,152.700
C01677=1088.636,-66.753,-52.501,174.595,17.006,152.700
C01678=1088.631,-67.002,-52.490,174.593,17.005,152.700
C01679=1088.624,-67.252,-52.478,174.592,17.004,152.701
C01680=1088.619,-67.502,-52.468,174.590,17.002,152.701
C01681=1088.614,-67.752,-52.456,174.589,17.001,152.701
C01682=1088.607,-68.002,-52.445,174.587,17.000,152.701
C01683=1088.601,-68.251,-52.434,174.585,16.999,152.701
C01684=1088.595,-68.500,-52.422,174.584,16.997,152.701
C01685=1088.589,-68.750,-52.411,174.582,16.996,152.701
C01686=1088.583,-69.000,-52.400,174.581,16.995,152.701
C01687=1088.578,-69.249,-52.389,174.579,16.994,152.701
C01688=1088.572,-69.499,-52.379,174.578,16.992,152.701
C01689=1088.566,-69.749,-52.367,174.576,16.991,152.701
C01690=1088.560,-69.998,-52.356,174.575,16.990,152.701
C01691=1088.554,-70.248,-52.346,174.573,16.989,152.701
C01692=1088.548,-70.498,-52.334,174.572,16.987,152.701
C01693=1088.543,-70.748,-52.323,174.570,16.986,152.701
C01694=1088.537,-70.997,-52.312,174.568,16.985,152.702
C01695=1088.531,-71.248,-52.301,174.567,16.984,152.702
C01696=1088.525,-71.497,-52.290,174.565,16.982,152.702
C01697=1088.519,-71.746,-52.278,174.564,16.981,152.702
C01698=1088.513,-71.995,-52.267,174.562,16.980,152.702
C01699=1088.507,-72.246,-52.256,174.560,16.979,152.702
C01700=1088.501,-72.495,-52.245,174.559,16.978,152.702
C01701=1088.495,-72.745,-52.234,174.557,16.976,152.702
C01702=1088.490,-72.994,-52.223,174.556,16.975,152.702
C01703=1088.483,-73.244,-52.212,174.555,16.975,152.702
C01704=1088.477,-73.494,-52.201,174.553,16.974,152.702
C01705=1088.472,-73.744,-52.191,174.552,16.972,152.702
C01706=1088.466,-73.993,-52.180,174.550,16.971,152.702
C01707=1088.460,-74.244,-52.169,174.549,16.970,152.703
C01708=1088.454,-74.493,-52.158,174.547,16.969,152.703
C01709=1088.448,-74.743,-52.147,174.545,16.968,152.703
C01710=1088.442,-74.993,-52.136,174.544,16.967,152.703
C01711=1088.436,-75.242,-52.125,174.542,16.966,152.703
C01712=1088.431,-75.492,-52.114,174.541,16.964,152.703
C01713=1088.424,-75.742,-52.104,174.539,16.963,152.703
C01714=1088.418,-75.991,-52.093,174.537,16.962,152.703
C01715=1088.412,-76.241,-52.082,174.536,16.961,152.703
C01716=1088.406,-76.490,-52.071,174.534,16.960,152.703
C01717=1088.400,-76.740,-52.060,174.533,16.958,152.703
C01718=1088.394,-76.990,-52.049,174.532,16.958,152.704
C01719=1088.388,-77.239,-52.039,174.530,16.957,152.704
C01720=1088.382,-77.488,-52.028,174.528,16.956,152.704
C01721=1088.376,-77.739,-52.017,174.527,16.954,152.704
C01722=1088.370,-77.989,-52.006,174.525,16.953,152.704
C01723=1088.365,-78.238,-51.995,174.524,16.952,152.704
C01724=1088.359,-78.488,-51.985,174.522,16.951,152.704
C01725=1088.352,-78.738,-51.974,174.521,16.950,152.704
C01726=1088.346,-78.987,-51.963,174.519,16.949,152.704
C01727=1088.340,-79.237,-51.952,174.517,16.947,152.704
C01728=1088.335,-79.487,-51.942,174.516,16.946,152.704
C01729=1088.328,-79.737,-51.931,174.514,16.945,152.705
C01730=1088.323,-79.986,-51.920,174.513,16.945,152.705
C01731=1088.316,-80.236,-51.910,174.512,16.944,152.705
C01732=1088.311,-80.485,-51.899,174.510,16.943,152.705
C01733=1088.304,-80.760,-51.887,174.508,16.941,152.705
C01734=1088.297,-81.035,-51.876,174.507,16.940,152.705
C01735=1088.291,-81.309,-51.864,174.504,16.939,152.705
C01736=1088.283,-81.583,-51.852,174.503,16.938,152.705
C01737=1088.278,-81.833,-51.842,174.501,16.936,152.705
C01738=1088.272,-82.082,-51.831,174.500,16.936,152.706
C01739=1088.265,-82.332,-51.820,174.499,16.935,152.706
C01740=1088.259,-82.582,-51.810,174.497,16.934,152.706
C01741=1088.253,-82.831,-51.799,174.495,16.933,152.706
C01742=1088.247,-83.081,-51.789,174.494,16.932,152.706
C01743=1088.241,-83.331,-51.778,174.492,16.930,152.706
C01744=1088.235,-83.581,-51.767,174.490,16.929,152.706
C01745=1088.228,-83.830,-51.757,174.489,16.928,152.706
C01746=1088.223,-84.080,-51.747,174.487,16.927,152.706
C01747=1088.216,-84.330,-51.736,174.486,16.927,152.706
C01748=1088.210,-84.579,-51.725,174.485,16.925,152.707
C01749=1088.205,-84.830,-51.715,174.483,16.924,152.707
C01750=1088.198,-85.079,-51.705,174.481,16.923,152.707
C01751=1088.193,-85.328,-51.694,174.480,16.922,152.707
C01752=1088.186,-85.579,-51.684,174.478,16.921,152.707
C01753=1088.180,-85.828,-51.673,174.476,16.920,152.707
C01754=1088.174,-86.078,-51.662,174.475,16.919,152.707
C01755=1088.168,-86.327,-51.652,174.474,16.918,152.707
C01756=1088.162,-86.577,-51.642,174.472,16.917,152.707
C01757=1088.155,-86.827,-51.631,174.471,16.916,152.707
C01758=1088.150,-87.077,-51.621,174.469,16.915,152.708
C01759=1088.144,-87.326,-51.610,174.467,16.914,152.708
C01760=1088.138,-87.576,-51.600,174.466,16.913,152.708
C01761=1088.132,-87.826,-51.589,174.464,16.912,152.708
C01762=1088.125,-88.076,-51.579,174.462,16.911,152.708
C01763=1088.119,-88.325,-51.568,174.461,16.911,152.708
C01764=1088.113,-88.575,-51.558,174.460,16.910,152.708
C01765=1088.108,-88.824,-51.547,174.458,16.908,152.708
C01766=1088.102,-89.075,-51.537,174.457,16.907,152.709
C01767=1088.096,-89.324,-51.527,174.455,16.906,152.709
C01768=1088.090,-89.573,-51.516,174.453,16.905,152.709
C01769=1088.083,-89.824,-51.506,174.452,16.904,152.709
C01770=1088.077,-90.073,-51.495,174.451,16.903,152.709
C01771=1088.071,-90.323,-51.486,174.449,16.902,152.709
C01772=1088.065,-90.572,-51.475,174.448,16.901,152.709
C01773=1088.059,-90.822,-51.465,174.446,16.901,152.709
C01774=1088.054,-91.072,-51.454,174.444,16.900,152.710
C01775=1088.047,-91.321,-51.444,174.442,16.898,152.710
C01776=1088.042,-91.571,-51.434,174.442,16.898,152.710
C01777=1088.035,-91.821,-51.423,174.440,16.897,152.710
C01778=1088.029,-92.071,-51.413,174.438,16.896,152.710
C01779=1088.023,-92.321,-51.402,174.437,16.895,152.710
C01780=1088.017,-92.570,-51.393,174.435,16.894,152.710
C01781=1088.011,-92.820,-51.382,174.433,16.892,152.710
C01782=1088.005,-93.070,-51.372,174.431,16.892,152.711
C01783=1088.000,-93.319,-51.361,174.431,16.891,152.711
C01784=1087.993,-93.569,-51.352,174.429,16.890,152.711
C01785=1087.988,-93.818,-51.341,174.427,16.889,152.711
C01786=1087.981,-94.068,-51.331,174.426,16.888,152.711
C01787=1087.976,-94.318,-51.321,174.424,16.887,152.711
C01788=1087.969,-94.568,-51.311,174.422,16.886,152.711
C01789=1087.963,-94.818,-51.300,174.422,16.885,152.711
C01790=1087.957,-95.067,-51.290,174.420,16.885,152.712
C01791=1087.952,-95.318,-51.280,174.418,16.884,152.712
C01792=1087.945,-95.567,-51.270,174.416,16.882,152.712
C01793=1087.940,-95.817,-51.260,174.415,16.881,152.712
C01794=1087.933,-96.066,-51.249,174.414,16.881,152.712
C01795=1087.928,-96.316,-51.239,174.412,16.880,152.712
C01796=1087.921,-96.565,-51.229,174.410,16.879,152.712
C01797=1087.915,-96.842,-51.218,174.409,16.878,152.712
C01798=1087.908,-97.119,-51.207,174.407,16.877,152.713
C01799=1087.902,-97.396,-51.195,174.406,16.876,152.713
C01800=1087.895,-97.673,-51.184,174.404,16.875,152.713
C01801=1087.889,-97.922,-51.174,174.402,16.874,152.713
C01802=1087.883,-98.172,-51.164,174.400,16.873,152.713
C01803=1087.877,-98.422,-51.154,174.399,16.872,152.713
C01804=1087.871,-98.671,-51.144,174.398,16.871,152.713
C01805=1087.865,-98.921,-51.134,174.396,16.871,152.714
C01806=1087.859,-99.170,-51.124,174.394,16.870,152.714
C01807=1087.853,-99.420,-51.114,174.393,16.869,152.714
C01808=1087.846,-99.671,-51.104,174.391,16.868,152.714
C01809=1087.840,-99.920,-51.094,174.390,16.867,152.714
C01810=1087.834,-100.170,-51.084,174.388,16.866,152.714
C01811=1087.828,-100.420,-51.074,174.387,16.865,152.714
C01812=1087.821,-100.669,-51.064,174.385,16.864,152.714
C01813=1087.816,-100.919,-51.054,174.383,16.864,152.715
C01814=1087.810,-101.169,-51.044,174.382,16.863,152.715
C01815=1087.804,-101.418,-51.034,174.381,16.862,152.715
C01816=1087.797,-101.668,-51.024,174.379,16.861,152.715
C01817=1087.792,-101.918,-51.014,174.377,16.860,152.715
C01818=1087.786,-102.168,-51.004,174.376,16.860,152.715
